KUKA KRL program: f1_Kuka_APT214T03S14.SRC

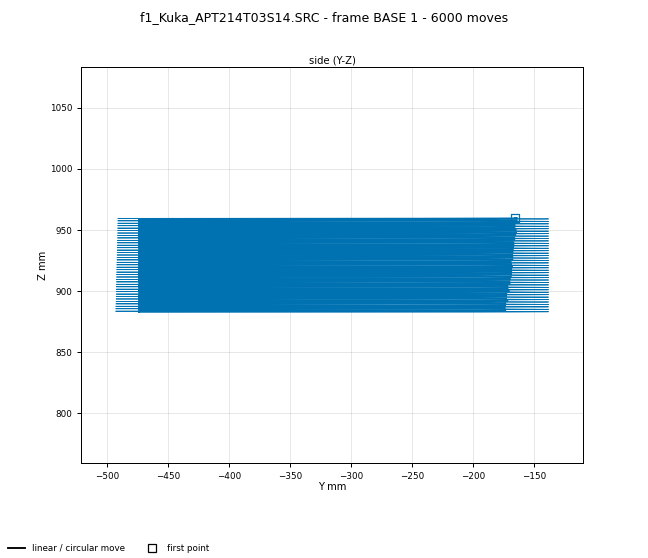
[picture p0: tool path of f1_Kuka_APT214T03S14.SRC in frame BASE 1, 6000 of 6001 moves have a stored position in this frame; points joined in program order, loops and branches not executed]
&ACCESS RVP
&REL 2
&PARAM TEMPLATE = C:\KRC\Roboter\Template\vorgabe
&PARAM EDITMASK = *
DEF f1_Kuka_APT214T03S14()


;FOLD INI;%{PE}%V3.2.0,%MKUKATPBASIS,%CINIT,%VCOMMON,%P
  ;FOLD BAS INI;%{E}%V3.2.0,%MKUKATPBASIS,%CINIT,%VINIT,%P
    GLOBAL INTERRUPT DECL 3 WHEN $STOPMESS==TRUE DO IR_STOPM ( )
    INTERRUPT ON 3
    BAS (#INITMOV,0 )
  ;ENDFOLD (BAS INI)
  ;FOLD USER INI;%{E}%V3.2.0,%MKUKATPUSER,%CINIT,%VINIT,%P
    ;Make your modifications here
  ;ENDFOLD (USER INI)
;ENDFOLD (INI)


;*** Make Null PTP Move
  PTP $pos_act

;*** Auto Load The Correct TOOL Data
  $tool=tool_data[3]

;*** Auto Load The Correct BASE Data
  $base=base_data[1]

  $ADVANCE = 5

;*** Restate Last Velocity
MMPM(30000.0)
SetRPM(6000)
LIN {X -0.031,Y -166.168,Z 960.065,A 0.000,B 0.000,C 90.000,E1 11.658} C_DIS
LIN {X 0.050,Y -163.859,Z 960.031,A 0.000,B 0.000,C 90.000,E1 5.511} C_DIS
LIN {X 0.017,Y -164.871,Z 959.968,A 0.000,B 0.000,C 90.000,E1 354.261} C_DIS
LIN {X -0.078,Y -167.650,Z 959.939,A 0.000,B 0.000,C 90.000,E1 349.050} C_DIS
LIN {X -0.007,Y -171.184,Z 959.915,A 0.000,B 0.000,C 90.000,E1 344.685} C_DIS
LIN {X 0.034,Y -175.840,Z 959.891,A 0.000,B 0.000,C 90.000,E1 340.369} C_DIS
LIN {X -0.004,Y -180.404,Z 959.872,A 0.000,B 0.000,C 90.000,E1 336.975} C_DIS
LIN {X 0.045,Y -185.731,Z 959.853,A 0.000,B 0.000,C 90.000,E1 333.589} C_DIS
LIN {X 0.060,Y -191.719,Z 959.835,A 0.000,B 0.000,C 90.000,E1 330.255} C_DIS
LIN {X -0.013,Y -198.321,Z 959.817,A 0.000,B 0.000,C 90.000,E1 326.993} C_DIS
LIN {X 0.015,Y -205.507,Z 959.799,A 0.000,B 0.000,C 90.000,E1 323.749} C_DIS
LIN {X -0.070,Y -214.244,Z 959.779,A 0.000,B 0.000,C 90.000,E1 320.194} C_DIS
LIN {X 0.036,Y -223.799,Z 959.759,A 0.000,B 0.000,C 90.000,E1 316.662} C_DIS
LIN {X -0.127,Y -232.037,Z 959.744,A 0.000,B 0.000,C 90.000,E1 314.028} C_DIS
LIN {X 0.056,Y -241.361,Z 959.730,A 0.000,B 0.000,C 90.000,E1 311.353} C_DIS
LIN {X 0.001,Y -250.281,Z 959.718,A 0.000,B 0.000,C 90.000,E1 309.152} C_DIS
LIN {X -0.109,Y -258.596,Z 959.707,A 0.000,B 0.000,C 90.000,E1 307.363} C_DIS
LIN {X 0.141,Y -271.571,Z 959.694,A 0.000,B 0.000,C 90.000,E1 304.818} C_DIS
LIN {X -0.058,Y -289.760,Z 959.676,A 0.000,B 0.000,C 90.000,E1 301.750} C_DIS
LIN {X -0.100,Y -304.933,Z 959.663,A 0.000,B 0.000,C 90.000,E1 299.411} C_DIS
LIN {X -0.098,Y -321.503,Z 959.651,A 0.000,B 0.000,C 90.000,E1 297.129} C_DIS
LIN {X -0.106,Y -334.635,Z 959.642,A 0.000,B 0.000,C 90.000,E1 295.540} C_DIS
LIN {X -0.116,Y -358.818,Z 959.627,A 0.000,B 0.000,C 90.000,E1 292.898} C_DIS
LIN {X -0.081,Y -377.767,Z 959.616,A 0.000,B 0.000,C 90.000,E1 290.972} C_DIS
LIN {X -0.056,Y -393.711,Z 959.608,A 0.000,B 0.000,C 90.000,E1 289.396} C_DIS
LIN {X -0.107,Y -404.139,Z 959.602,A 0.000,B 0.000,C 90.000,E1 288.362} C_DIS
LIN {X 0.117,Y -414.354,Z 959.596,A 0.000,B 0.000,C 90.000,E1 287.275} C_DIS
LIN {X 0.081,Y -424.254,Z 959.590,A 0.000,B 0.000,C 90.000,E1 286.205} C_DIS
LIN {X 0.005,Y -433.708,Z 959.584,A 0.000,B 0.000,C 90.000,E1 285.134} C_DIS
LIN {X 0.038,Y -442.447,Z 959.578,A 0.000,B 0.000,C 90.000,E1 284.064} C_DIS
LIN {X 0.069,Y -450.785,Z 959.572,A 0.000,B 0.000,C 90.000,E1 283.008} C_DIS
LIN {X 0.028,Y -460.710,Z 959.565,A 0.000,B 0.000,C 90.000,E1 281.715} C_DIS
LIN {X -0.184,Y -468.269,Z 959.559,A 0.000,B 0.000,C 90.000,E1 280.715} C_DIS
LIN {X 0.202,Y -473.450,Z 959.555,A 0.000,B 0.000,C 90.000,E1 279.905} C_DIS
LIN {X 0.180,Y -478.073,Z 959.551,A 0.000,B 0.000,C 90.000,E1 279.151} C_DIS
LIN {X 0.195,Y -481.999,Z 959.547,A 0.000,B 0.000,C 90.000,E1 278.398} C_DIS
LIN {X -0.115,Y -484.263,Z 959.544,A 0.000,B 0.000,C 90.000,E1 277.936} C_DIS
LIN {X 0.131,Y -486.237,Z 959.541,A 0.000,B 0.000,C 90.000,E1 277.409} C_DIS
LIN {X -0.165,Y -487.852,Z 959.539,A 0.000,B 0.000,C 90.000,E1 276.947} C_DIS
LIN {X 0.034,Y -489.159,Z 959.536,A 0.000,B 0.000,C 90.000,E1 276.429} C_DIS
LIN {X 0.244,Y -490.135,Z 959.533,A 0.000,B 0.000,C 90.000,E1 275.910} C_DIS
LIN {X -0.074,Y -490.762,Z 959.530,A 0.000,B 0.000,C 90.000,E1 275.454} C_DIS
LIN {X 0.152,Y -491.016,Z 959.528,A 0.000,B 0.000,C 90.000,E1 274.935} C_DIS
LIN {X -0.111,Y -490.869,Z 959.525,A 0.000,B 0.000,C 90.000,E1 274.473} C_DIS
LIN {X 0.114,Y -490.251,Z 959.522,A 0.000,B 0.000,C 90.000,E1 273.955} C_DIS
LIN {X -0.183,Y -489.140,Z 959.519,A 0.000,B 0.000,C 90.000,E1 273.498} C_DIS
LIN {X 0.034,Y -487.440,Z 959.517,A 0.000,B 0.000,C 90.000,E1 272.980} C_DIS
LIN {X 0.217,Y -485.143,Z 959.514,A 0.000,B 0.000,C 90.000,E1 272.465} C_DIS
LIN {X -0.095,Y -482.097,Z 959.511,A 0.000,B 0.000,C 90.000,E1 272.007} C_DIS
LIN {X 0.074,Y -478.192,Z 959.508,A 0.000,B 0.000,C 90.000,E1 271.489} C_DIS
LIN {X 0.207,Y -473.231,Z 959.506,A 0.000,B 0.000,C 90.000,E1 270.974} C_DIS
LIN {X 0.022,Y -467.466,Z 959.503,A 0.000,B 0.000,C 90.000,E1 270.516} C_DIS
LIN {X -0.191,Y -461.347,Z 959.500,A 0.000,B 0.000,C 90.000,E1 270.115} C_DIS
LIN {X -0.006,Y -454.864,Z 959.498,A 0.000,B 0.000,C 90.000,E1 269.714} C_DIS
LIN {X 0.154,Y -448.019,Z 959.497,A 0.000,B 0.000,C 90.000,E1 269.370} C_DIS
LIN {X -0.150,Y -441.116,Z 959.495,A 0.000,B 0.000,C 90.000,E1 269.141} C_DIS
LIN {X -0.111,Y -433.920,Z 959.494,A 0.000,B 0.000,C 90.000,E1 268.912} C_DIS
LIN {X -0.201,Y -426.014,Z 959.493,A 0.000,B 0.000,C 90.000,E1 268.740} C_DIS
LIN {X 0.015,Y -417.851,Z 959.492,A 0.000,B 0.000,C 90.000,E1 268.568} C_DIS
LIN {X -0.140,Y -410.678,Z 959.492,A 0.000,B 0.000,C 90.000,E1 268.511} C_DIS
LIN {X -0.033,Y -402.201,Z 959.491,A 0.000,B 0.000,C 90.000,E1 268.453} C_DIS
LIN {X -0.040,Y -181.202,Z 959.491,A 0.000,B 0.000,C 90.000,E1 268.453} C_DIS
LIN {X 0.070,Y -180.868,Z 959.472,A 0.000,B 0.000,C 90.000,E1 265.008} C_DIS
LIN {X -0.054,Y -178.983,Z 959.444,A 0.000,B 0.000,C 90.000,E1 259.982} C_DIS
LIN {X -0.042,Y -177.958,Z 959.435,A 0.000,B 0.000,C 90.000,E1 258.285} C_DIS
LIN {X -0.022,Y -175.600,Z 959.411,A 0.000,B 0.000,C 90.000,E1 254.031} C_DIS
LIN {X -0.009,Y -172.324,Z 959.388,A 0.000,B 0.000,C 90.000,E1 249.752} C_DIS
LIN {X -0.031,Y -171.801,Z 959.383,A 0.000,B 0.000,C 90.000,E1 248.901} C_DIS
LIN {X 0.006,Y -169.476,Z 959.368,A 0.000,B 0.000,C 90.000,E1 246.305} C_DIS
LIN {X -0.087,Y -166.803,Z 959.349,A 0.000,B 0.000,C 90.000,E1 242.871} C_DIS
LIN {X 0.056,Y -162.783,Z 959.325,A 0.000,B 0.000,C 90.000,E1 238.456} C_DIS
LIN {X 0.032,Y -161.472,Z 959.315,A 0.000,B 0.000,C 90.000,E1 236.707} C_DIS
LIN {X 0.073,Y -157.467,Z 959.291,A 0.000,B 0.000,C 90.000,E1 232.271} C_DIS
LIN {X 0.005,Y -155.481,Z 959.276,A 0.000,B 0.000,C 90.000,E1 229.622} C_DIS
LIN {X -0.062,Y -151.789,Z 959.251,A 0.000,B 0.000,C 90.000,E1 225.162} C_DIS
LIN {X -0.048,Y -149.998,Z 959.236,A 0.000,B 0.000,C 90.000,E1 222.447} C_DIS
LIN {X -0.017,Y -146.827,Z 959.210,A 0.000,B 0.000,C 90.000,E1 217.890} C_DIS
LIN {X -0.030,Y -145.407,Z 959.195,A 0.000,B 0.000,C 90.000,E1 215.152} C_DIS
LIN {X 0.005,Y -142.839,Z 959.170,A 0.000,B 0.000,C 90.000,E1 210.541} C_DIS
LIN {X -0.064,Y -141.452,Z 959.149,A 0.000,B 0.000,C 90.000,E1 206.873} C_DIS
LIN {X -0.025,Y -139.372,Z 959.113,A 0.000,B 0.000,C 90.000,E1 200.355} C_DIS
LIN {X -0.082,Y -138.821,Z 959.097,A 0.000,B 0.000,C 90.000,E1 197.583} C_DIS
LIN {X 0.007,Y -138.352,Z 959.056,A 0.000,B 0.000,C 90.000,E1 190.074} C_DIS
LIN {X -0.021,Y -139.534,Z 959.004,A 0.000,B 0.000,C 90.000,E1 180.745} C_DIS
LIN {X 0.072,Y -141.217,Z 958.973,A 0.000,B 0.000,C 90.000,E1 175.122} C_DIS
LIN {X 0.032,Y -142.591,Z 958.958,A 0.000,B 0.000,C 90.000,E1 172.356} C_DIS
LIN {X -0.014,Y -144.891,Z 958.932,A 0.000,B 0.000,C 90.000,E1 167.757} C_DIS
LIN {X -0.062,Y -147.519,Z 958.912,A 0.000,B 0.000,C 90.000,E1 164.102} C_DIS
LIN {X 0.013,Y -150.113,Z 958.891,A 0.000,B 0.000,C 90.000,E1 160.423} C_DIS
LIN {X 0.025,Y -153.473,Z 958.871,A 0.000,B 0.000,C 90.000,E1 156.794} C_DIS
LIN {X 0.015,Y -157.838,Z 958.846,A 0.000,B 0.000,C 90.000,E1 152.308} C_DIS
LIN {X 0.046,Y -162.122,Z 958.826,A 0.000,B 0.000,C 90.000,E1 148.742} C_DIS
LIN {X -0.069,Y -166.324,Z 958.807,A 0.000,B 0.000,C 90.000,E1 145.261} C_DIS
LIN {X 0.032,Y -171.341,Z 958.788,A 0.000,B 0.000,C 90.000,E1 141.743} C_DIS
LIN {X -0.041,Y -176.244,Z 958.768,A 0.000,B 0.000,C 90.000,E1 138.324} C_DIS
LIN {X 0.079,Y -180.525,Z 958.754,A 0.000,B 0.000,C 90.000,E1 135.729} C_DIS
LIN {X 0.059,Y -185.928,Z 958.735,A 0.000,B 0.000,C 90.000,E1 132.366} C_DIS
LIN {X -0.007,Y -190.558,Z 958.722,A 0.000,B 0.000,C 90.000,E1 129.886} C_DIS
LIN {X 0.020,Y -194.806,Z 958.708,A 0.000,B 0.000,C 90.000,E1 127.397} C_DIS
LIN {X -0.006,Y -297.968,Z 958.708,A 0.000,B 0.000,C 90.000,E1 127.397} C_DIS
LIN {X -0.109,Y -300.519,Z 958.707,A 0.000,B 0.000,C 90.000,E1 127.363} C_DIS
LIN {X -0.014,Y -304.144,Z 958.706,A 0.000,B 0.000,C 90.000,E1 127.156} C_DIS
LIN {X 0.086,Y -306.383,Z 958.705,A 0.000,B 0.000,C 90.000,E1 126.950} C_DIS
LIN {X 0.037,Y -309.504,Z 958.703,A 0.000,B 0.000,C 90.000,E1 126.583} C_DIS
LIN {X -0.163,Y -311.442,Z 958.701,A 0.000,B 0.000,C 90.000,E1 126.297} C_DIS
LIN {X 0.072,Y -312.952,Z 958.700,A 0.000,B 0.000,C 90.000,E1 125.931} C_DIS
LIN {X -0.087,Y -315.137,Z 958.696,A 0.000,B 0.000,C 90.000,E1 125.311} C_DIS
LIN {X 0.037,Y -325.779,Z 958.678,A 0.000,B 0.000,C 90.000,E1 122.084} C_DIS
LIN {X -0.132,Y -336.713,Z 958.663,A 0.000,B 0.000,C 90.000,E1 119.283} C_DIS
LIN {X -0.033,Y -349.037,Z 958.647,A 0.000,B 0.000,C 90.000,E1 116.488} C_DIS
LIN {X -0.038,Y -362.857,Z 958.632,A 0.000,B 0.000,C 90.000,E1 113.770} C_DIS
LIN {X -0.051,Y -376.497,Z 958.619,A 0.000,B 0.000,C 90.000,E1 111.408} C_DIS
LIN {X 0.003,Y -391.515,Z 958.606,A 0.000,B 0.000,C 90.000,E1 109.087} C_DIS
LIN {X -0.201,Y -408.016,Z 958.594,A 0.000,B 0.000,C 90.000,E1 106.858} C_DIS
LIN {X -0.131,Y -426.122,Z 958.581,A 0.000,B 0.000,C 90.000,E1 104.647} C_DIS
LIN {X -0.199,Y -445.757,Z 958.570,A 0.000,B 0.000,C 90.000,E1 102.535} C_DIS
LIN {X 0.059,Y -466.092,Z 958.559,A 0.000,B 0.000,C 90.000,E1 100.546} C_DIS
LIN {X 0.072,Y -468.438,Z 958.557,A 0.000,B 0.000,C 90.000,E1 100.310} C_DIS
LIN {X -0.026,Y -470.296,Z 958.556,A 0.000,B 0.000,C 90.000,E1 100.074} C_DIS
LIN {X -0.207,Y -471.699,Z 958.555,A 0.000,B 0.000,C 90.000,E1 99.849} C_DIS
LIN {X -0.031,Y -473.539,Z 958.552,A 0.000,B 0.000,C 90.000,E1 99.321} C_DIS
LIN {X 0.077,Y -474.283,Z 958.549,A 0.000,B 0.000,C 90.000,E1 98.803} C_DIS
LIN {X 0.268,Y -474.059,Z 958.546,A 0.000,B 0.000,C 90.000,E1 98.276} C_DIS
LIN {X -0.077,Y -472.835,Z 958.543,A 0.000,B 0.000,C 90.000,E1 97.814} C_DIS
LIN {X 0.188,Y -471.792,Z 958.542,A 0.000,B 0.000,C 90.000,E1 97.530} C_DIS
LIN {X 0.047,Y -470.392,Z 958.541,A 0.000,B 0.000,C 90.000,E1 97.296} C_DIS
LIN {X 0.100,Y -458.658,Z 958.531,A 0.000,B 0.000,C 90.000,E1 95.511} C_DIS
LIN {X 0.121,Y -445.384,Z 958.519,A 0.000,B 0.000,C 90.000,E1 93.440} C_DIS
LIN {X 0.105,Y -428.779,Z 958.505,A 0.000,B 0.000,C 90.000,E1 90.802} C_DIS
LIN {X 0.128,Y -411.902,Z 958.488,A 0.000,B 0.000,C 90.000,E1 87.822} C_DIS
LIN {X 0.175,Y -402.774,Z 958.479,A 0.000,B 0.000,C 90.000,E1 86.159} C_DIS
LIN {X 0.131,Y -392.001,Z 958.468,A 0.000,B 0.000,C 90.000,E1 84.204} C_DIS
LIN {X -0.067,Y -382.677,Z 958.458,A 0.000,B 0.000,C 90.000,E1 82.527} C_DIS
LIN {X -0.047,Y -373.069,Z 958.449,A 0.000,B 0.000,C 90.000,E1 80.792} C_DIS
LIN {X -0.148,Y -363.193,Z 958.439,A 0.000,B 0.000,C 90.000,E1 79.050} C_DIS
LIN {X 0.066,Y -353.138,Z 958.429,A 0.000,B 0.000,C 90.000,E1 77.229} C_DIS
LIN {X -0.090,Y -338.180,Z 958.414,A 0.000,B 0.000,C 90.000,E1 74.519} C_DIS
LIN {X 0.039,Y -324.200,Z 958.398,A 0.000,B 0.000,C 90.000,E1 71.692} C_DIS
LIN {X -0.036,Y -312.152,Z 958.384,A 0.000,B 0.000,C 90.000,E1 69.156} C_DIS
LIN {X 0.027,Y -301.623,Z 958.372,A 0.000,B 0.000,C 90.000,E1 66.869} C_DIS
LIN {X 0.094,Y -291.227,Z 958.359,A 0.000,B 0.000,C 90.000,E1 64.537} C_DIS
LIN {X 0.061,Y -280.913,Z 958.346,A 0.000,B 0.000,C 90.000,E1 62.180} C_DIS
LIN {X -0.046,Y -270.635,Z 958.332,A 0.000,B 0.000,C 90.000,E1 59.793} C_DIS
LIN {X 0.050,Y -259.319,Z 958.317,A 0.000,B 0.000,C 90.000,E1 56.962} C_DIS
LIN {X -0.049,Y -247.134,Z 958.299,A 0.000,B 0.000,C 90.000,E1 53.749} C_DIS
LIN {X -0.049,Y -235.992,Z 958.280,A 0.000,B 0.000,C 90.000,E1 50.436} C_DIS
LIN {X 0.050,Y -225.633,Z 958.261,A 0.000,B 0.000,C 90.000,E1 47.025} C_DIS
LIN {X 0.088,Y -217.040,Z 958.244,A 0.000,B 0.000,C 90.000,E1 43.947} C_DIS
LIN {X -0.045,Y -208.949,Z 958.227,A 0.000,B 0.000,C 90.000,E1 40.862} C_DIS
LIN {X -0.029,Y -201.480,Z 958.209,A 0.000,B 0.000,C 90.000,E1 37.684} C_DIS
LIN {X -0.008,Y -194.630,Z 958.191,A 0.000,B 0.000,C 90.000,E1 34.452} C_DIS
LIN {X -0.013,Y -188.415,Z 958.173,A 0.000,B 0.000,C 90.000,E1 31.180} C_DIS
LIN {X 0.030,Y -182.953,Z 958.155,A 0.000,B 0.000,C 90.000,E1 27.847} C_DIS
LIN {X -0.062,Y -178.106,Z 958.136,A 0.000,B 0.000,C 90.000,E1 24.515} C_DIS
LIN {X -0.015,Y -173.074,Z 958.112,A 0.000,B 0.000,C 90.000,E1 20.248} C_DIS
LIN {X -0.032,Y -169.140,Z 958.089,A 0.000,B 0.000,C 90.000,E1 15.953} C_DIS
LIN {X 0.039,Y -166.285,Z 958.064,A 0.000,B 0.000,C 90.000,E1 11.591} C_DIS
LIN {X -0.070,Y -163.987,Z 958.030,A 0.000,B 0.000,C 90.000,E1 5.511} C_DIS
LIN {X 0.023,Y -165.053,Z 957.968,A 0.000,B 0.000,C 90.000,E1 354.261} C_DIS
LIN {X -0.065,Y -167.841,Z 957.939,A 0.000,B 0.000,C 90.000,E1 349.050} C_DIS
LIN {X -0.032,Y -171.390,Z 957.915,A 0.000,B 0.000,C 90.000,E1 344.700} C_DIS
LIN {X 0.061,Y -176.062,Z 957.891,A 0.000,B 0.000,C 90.000,E1 340.369} C_DIS
LIN {X 0.028,Y -180.646,Z 957.872,A 0.000,B 0.000,C 90.000,E1 336.975} C_DIS
LIN {X -0.082,Y -185.957,Z 957.853,A 0.000,B 0.000,C 90.000,E1 333.640} C_DIS
LIN {X 0.012,Y -191.932,Z 957.835,A 0.000,B 0.000,C 90.000,E1 330.284} C_DIS
LIN {X 0.040,Y -198.523,Z 957.817,A 0.000,B 0.000,C 90.000,E1 326.993} C_DIS
LIN {X -0.045,Y -205.728,Z 957.799,A 0.000,B 0.000,C 90.000,E1 323.783} C_DIS
LIN {X -0.039,Y -213.425,Z 957.781,A 0.000,B 0.000,C 90.000,E1 320.598} C_DIS
LIN {X 0.041,Y -222.894,Z 957.762,A 0.000,B 0.000,C 90.000,E1 317.067} C_DIS
LIN {X -0.042,Y -232.250,Z 957.745,A 0.000,B 0.000,C 90.000,E1 314.028} C_DIS
LIN {X 0.133,Y -242.974,Z 957.728,A 0.000,B 0.000,C 90.000,E1 310.987} C_DIS
LIN {X -0.081,Y -252.062,Z 957.716,A 0.000,B 0.000,C 90.000,E1 308.830} C_DIS
LIN {X 0.001,Y -258.762,Z 957.708,A 0.000,B 0.000,C 90.000,E1 307.363} C_DIS
LIN {X -0.120,Y -271.661,Z 957.694,A 0.000,B 0.000,C 90.000,E1 304.898} C_DIS
LIN {X 0.070,Y -289.797,Z 957.676,A 0.000,B 0.000,C 90.000,E1 301.750} C_DIS
LIN {X 0.035,Y -304.932,Z 957.663,A 0.000,B 0.000,C 90.000,E1 299.411} C_DIS
LIN {X 0.044,Y -321.401,Z 957.651,A 0.000,B 0.000,C 90.000,E1 297.129} C_DIS
LIN {X 0.062,Y -333.998,Z 957.642,A 0.000,B 0.000,C 90.000,E1 295.591} C_DIS
LIN {X 0.025,Y -358.052,Z 957.628,A 0.000,B 0.000,C 90.000,E1 292.950} C_DIS
LIN {X -0.067,Y -379.492,Z 957.615,A 0.000,B 0.000,C 90.000,E1 290.791} C_DIS
LIN {X 0.028,Y -392.885,Z 957.608,A 0.000,B 0.000,C 90.000,E1 289.450} C_DIS
LIN {X -0.063,Y -403.354,Z 957.602,A 0.000,B 0.000,C 90.000,E1 288.417} C_DIS
LIN {X 0.130,Y -413.596,Z 957.596,A 0.000,B 0.000,C 90.000,E1 287.330} C_DIS
LIN {X 0.100,Y -423.566,Z 957.590,A 0.000,B 0.000,C 90.000,E1 286.260} C_DIS
LIN {X 0.017,Y -433.028,Z 957.584,A 0.000,B 0.000,C 90.000,E1 285.190} C_DIS
LIN {X 0.040,Y -441.816,Z 957.578,A 0.000,B 0.000,C 90.000,E1 284.120} C_DIS
LIN {X -0.135,Y -452.195,Z 957.571,A 0.000,B 0.000,C 90.000,E1 282.827} C_DIS
LIN {X -0.169,Y -462.102,Z 957.564,A 0.000,B 0.000,C 90.000,E1 281.535} C_DIS
LIN {X 0.003,Y -469.556,Z 957.558,A 0.000,B 0.000,C 90.000,E1 280.489} C_DIS
LIN {X 0.026,Y -474.604,Z 957.554,A 0.000,B 0.000,C 90.000,E1 279.726} C_DIS
LIN {X 0.005,Y -479.128,Z 957.550,A 0.000,B 0.000,C 90.000,E1 278.973} C_DIS
LIN {X 0.029,Y -482.897,Z 957.546,A 0.000,B 0.000,C 90.000,E1 278.219} C_DIS
LIN {X 0.082,Y -486.004,Z 957.542,A 0.000,B 0.000,C 90.000,E1 277.466} C_DIS
LIN {X -0.217,Y -487.679,Z 957.539,A 0.000,B 0.000,C 90.000,E1 277.004} C_DIS
LIN {X -0.019,Y -489.027,Z 957.536,A 0.000,B 0.000,C 90.000,E1 276.486} C_DIS
LIN {X 0.189,Y -490.059,Z 957.533,A 0.000,B 0.000,C 90.000,E1 275.967} C_DIS
LIN {X -0.130,Y -490.734,Z 957.531,A 0.000,B 0.000,C 90.000,E1 275.511} C_DIS
LIN {X 0.094,Y -491.036,Z 957.528,A 0.000,B 0.000,C 90.000,E1 274.992} C_DIS
LIN {X -0.168,Y -490.957,Z 957.525,A 0.000,B 0.000,C 90.000,E1 274.531} C_DIS
LIN {X 0.056,Y -490.405,Z 957.522,A 0.000,B 0.000,C 90.000,E1 274.012} C_DIS
LIN {X -0.241,Y -489.317,Z 957.520,A 0.000,B 0.000,C 90.000,E1 273.555} C_DIS
LIN {X -0.022,Y -487.729,Z 957.517,A 0.000,B 0.000,C 90.000,E1 273.037} C_DIS
LIN {X -0.174,Y -486.739,Z 957.516,A 0.000,B 0.000,C 90.000,E1 272.808} C_DIS
LIN {X 0.006,Y -484.152,Z 957.513,A 0.000,B 0.000,C 90.000,E1 272.293} C_DIS
LIN {X 0.187,Y -480.765,Z 957.510,A 0.000,B 0.000,C 90.000,E1 271.776} C_DIS
LIN {X -0.146,Y -476.527,Z 957.507,A 0.000,B 0.000,C 90.000,E1 271.318} C_DIS
LIN {X 0.044,Y -471.215,Z 957.504,A 0.000,B 0.000,C 90.000,E1 270.802} C_DIS
LIN {X 0.021,Y -465.321,Z 957.502,A 0.000,B 0.000,C 90.000,E1 270.344} C_DIS
LIN {X -0.054,Y -459.128,Z 957.500,A 0.000,B 0.000,C 90.000,E1 269.943} C_DIS
LIN {X -0.164,Y -452.517,Z 957.498,A 0.000,B 0.000,C 90.000,E1 269.599} C_DIS
LIN {X 0.141,Y -445.677,Z 957.496,A 0.000,B 0.000,C 90.000,E1 269.255} C_DIS
LIN {X -0.057,Y -438.526,Z 957.495,A 0.000,B 0.000,C 90.000,E1 269.026} C_DIS
LIN {X 0.078,Y -431.034,Z 957.493,A 0.000,B 0.000,C 90.000,E1 268.797} C_DIS
LIN {X 0.090,Y -423.172,Z 957.492,A 0.000,B 0.000,C 90.000,E1 268.625} C_DIS
LIN {X -0.031,Y -414.503,Z 957.492,A 0.000,B 0.000,C 90.000,E1 268.511} C_DIS
LIN {X -0.027,Y -407.110,Z 957.491,A 0.000,B 0.000,C 90.000,E1 268.453} C_DIS
LIN {X -0.140,Y -402.934,Z 957.491,A 0.000,B 0.000,C 90.000,E1 268.453} C_DIS
LIN {X -0.088,Y -181.199,Z 957.491,A 0.000,B 0.000,C 90.000,E1 268.453} C_DIS
LIN {X 0.022,Y -180.865,Z 957.472,A 0.000,B 0.000,C 90.000,E1 265.008} C_DIS
LIN {X 0.075,Y -178.979,Z 957.444,A 0.000,B 0.000,C 90.000,E1 259.926} C_DIS
LIN {X 0.085,Y -177.948,Z 957.435,A 0.000,B 0.000,C 90.000,E1 258.229} C_DIS
LIN {X -0.069,Y -175.589,Z 957.411,A 0.000,B 0.000,C 90.000,E1 254.031} C_DIS
LIN {X -0.057,Y -172.315,Z 957.387,A 0.000,B 0.000,C 90.000,E1 249.752} C_DIS
LIN {X -0.078,Y -171.792,Z 957.383,A 0.000,B 0.000,C 90.000,E1 248.901} C_DIS
LIN {X -0.040,Y -169.462,Z 957.368,A 0.000,B 0.000,C 90.000,E1 246.305} C_DIS
LIN {X 0.016,Y -166.791,Z 957.349,A 0.000,B 0.000,C 90.000,E1 242.820} C_DIS
LIN {X 0.011,Y -162.771,Z 957.325,A 0.000,B 0.000,C 90.000,E1 238.456} C_DIS
LIN {X -0.012,Y -161.460,Z 957.315,A 0.000,B 0.000,C 90.000,E1 236.707} C_DIS
LIN {X 0.029,Y -157.454,Z 957.290,A 0.000,B 0.000,C 90.000,E1 232.271} C_DIS
LIN {X -0.038,Y -155.465,Z 957.276,A 0.000,B 0.000,C 90.000,E1 229.622} C_DIS
LIN {X 0.003,Y -151.779,Z 957.251,A 0.000,B 0.000,C 90.000,E1 225.121} C_DIS
LIN {X 0.019,Y -149.984,Z 957.236,A 0.000,B 0.000,C 90.000,E1 222.405} C_DIS
LIN {X -0.059,Y -146.817,Z 957.210,A 0.000,B 0.000,C 90.000,E1 217.890} C_DIS
LIN {X 0.046,Y -145.396,Z 957.195,A 0.000,B 0.000,C 90.000,E1 215.105} C_DIS
LIN {X -0.036,Y -142.832,Z 957.170,A 0.000,B 0.000,C 90.000,E1 210.541} C_DIS
LIN {X 0.021,Y -141.443,Z 957.149,A 0.000,B 0.000,C 90.000,E1 206.821} C_DIS
LIN {X 0.065,Y -139.369,Z 957.113,A 0.000,B 0.000,C 90.000,E1 200.301} C_DIS
LIN {X 0.051,Y -138.817,Z 957.097,A 0.000,B 0.000,C 90.000,E1 197.511} C_DIS
LIN {X -0.035,Y -138.352,Z 957.056,A 0.000,B 0.000,C 90.000,E1 190.074} C_DIS
LIN {X -0.062,Y -139.536,Z 957.004,A 0.000,B 0.000,C 90.000,E1 180.745} C_DIS
LIN {X 0.032,Y -141.225,Z 956.973,A 0.000,B 0.000,C 90.000,E1 175.122} C_DIS
LIN {X -0.010,Y -142.596,Z 956.958,A 0.000,B 0.000,C 90.000,E1 172.356} C_DIS
LIN {X -0.056,Y -144.901,Z 956.932,A 0.000,B 0.000,C 90.000,E1 167.757} C_DIS
LIN {X 0.038,Y -147.529,Z 956.911,A 0.000,B 0.000,C 90.000,E1 164.047} C_DIS
LIN {X -0.030,Y -150.127,Z 956.891,A 0.000,B 0.000,C 90.000,E1 160.423} C_DIS
LIN {X -0.019,Y -153.491,Z 956.871,A 0.000,B 0.000,C 90.000,E1 156.794} C_DIS
LIN {X 0.045,Y -157.855,Z 956.846,A 0.000,B 0.000,C 90.000,E1 152.281} C_DIS
LIN {X 0.001,Y -162.141,Z 956.826,A 0.000,B 0.000,C 90.000,E1 148.742} C_DIS
LIN {X -0.021,Y -166.345,Z 956.807,A 0.000,B 0.000,C 90.000,E1 145.229} C_DIS
LIN {X -0.015,Y -171.362,Z 956.787,A 0.000,B 0.000,C 90.000,E1 141.743} C_DIS
LIN {X -0.088,Y -176.268,Z 956.768,A 0.000,B 0.000,C 90.000,E1 138.324} C_DIS
LIN {X 0.031,Y -180.552,Z 956.754,A 0.000,B 0.000,C 90.000,E1 135.729} C_DIS
LIN {X 0.010,Y -185.954,Z 956.735,A 0.000,B 0.000,C 90.000,E1 132.366} C_DIS
LIN {X 0.066,Y -190.586,Z 956.721,A 0.000,B 0.000,C 90.000,E1 129.850} C_DIS
LIN {X -0.022,Y -194.746,Z 956.708,A 0.000,B 0.000,C 90.000,E1 127.443} C_DIS
LIN {X -0.088,Y -297.857,Z 956.708,A 0.000,B 0.000,C 90.000,E1 127.443} C_DIS
LIN {X -0.011,Y -299.609,Z 956.708,A 0.000,B 0.000,C 90.000,E1 127.397} C_DIS
LIN {X 0.080,Y -302.988,Z 956.707,A 0.000,B 0.000,C 90.000,E1 127.237} C_DIS
LIN {X -0.049,Y -306.366,Z 956.706,A 0.000,B 0.000,C 90.000,E1 126.996} C_DIS
LIN {X 0.110,Y -310.028,Z 956.703,A 0.000,B 0.000,C 90.000,E1 126.503} C_DIS
LIN {X -0.111,Y -311.840,Z 956.701,A 0.000,B 0.000,C 90.000,E1 126.217} C_DIS
LIN {X -0.081,Y -313.256,Z 956.699,A 0.000,B 0.000,C 90.000,E1 125.884} C_DIS
LIN {X -0.018,Y -324.881,Z 956.680,A 0.000,B 0.000,C 90.000,E1 122.339} C_DIS
LIN {X 0.067,Y -335.703,Z 956.664,A 0.000,B 0.000,C 90.000,E1 119.489} C_DIS
LIN {X -0.156,Y -347.901,Z 956.648,A 0.000,B 0.000,C 90.000,E1 116.744} C_DIS
LIN {X -0.056,Y -361.590,Z 956.633,A 0.000,B 0.000,C 90.000,E1 114.003} C_DIS
LIN {X -0.111,Y -375.105,Z 956.620,A 0.000,B 0.000,C 90.000,E1 111.642} C_DIS
LIN {X -0.103,Y -389.985,Z 956.607,A 0.000,B 0.000,C 90.000,E1 109.322} C_DIS
LIN {X 0.033,Y -406.340,Z 956.595,A 0.000,B 0.000,C 90.000,E1 107.040} C_DIS
LIN {X 0.074,Y -424.286,Z 956.582,A 0.000,B 0.000,C 90.000,E1 104.828} C_DIS
LIN {X 0.018,Y -443.817,Z 956.571,A 0.000,B 0.000,C 90.000,E1 102.703} C_DIS
LIN {X 0.144,Y -464.099,Z 956.560,A 0.000,B 0.000,C 90.000,E1 100.715} C_DIS
LIN {X 0.077,Y -466.659,Z 956.558,A 0.000,B 0.000,C 90.000,E1 100.489} C_DIS
LIN {X 0.095,Y -468.866,Z 956.557,A 0.000,B 0.000,C 90.000,E1 100.254} C_DIS
LIN {X -0.058,Y -470.658,Z 956.556,A 0.000,B 0.000,C 90.000,E1 100.018} C_DIS
LIN {X 0.251,Y -472.005,Z 956.554,A 0.000,B 0.000,C 90.000,E1 99.726} C_DIS
LIN {X -0.115,Y -473.691,Z 956.551,A 0.000,B 0.000,C 90.000,E1 99.265} C_DIS
LIN {X -0.004,Y -474.311,Z 956.549,A 0.000,B 0.000,C 90.000,E1 98.746} C_DIS
LIN {X 0.188,Y -473.964,Z 956.546,A 0.000,B 0.000,C 90.000,E1 98.219} C_DIS
LIN {X -0.156,Y -472.605,Z 956.543,A 0.000,B 0.000,C 90.000,E1 97.757} C_DIS
LIN {X 0.109,Y -471.478,Z 956.542,A 0.000,B 0.000,C 90.000,E1 97.473} C_DIS
LIN {X 0.079,Y -466.628,Z 956.537,A 0.000,B 0.000,C 90.000,E1 96.720} C_DIS
LIN {X -0.131,Y -453.282,Z 956.526,A 0.000,B 0.000,C 90.000,E1 94.702} C_DIS
LIN {X -0.191,Y -443.341,Z 956.517,A 0.000,B 0.000,C 90.000,E1 93.151} C_DIS
LIN {X 0.116,Y -422.154,Z 956.498,A 0.000,B 0.000,C 90.000,E1 89.656} C_DIS
LIN {X 0.109,Y -410.054,Z 956.486,A 0.000,B 0.000,C 90.000,E1 87.478} C_DIS
LIN {X 0.147,Y -400.864,Z 956.477,A 0.000,B 0.000,C 90.000,E1 85.812} C_DIS
LIN {X 0.078,Y -390.096,Z 956.466,A 0.000,B 0.000,C 90.000,E1 83.856} C_DIS
LIN {X -0.200,Y -380.695,Z 956.456,A 0.000,B 0.000,C 90.000,E1 82.186} C_DIS
LIN {X -0.161,Y -371.062,Z 956.447,A 0.000,B 0.000,C 90.000,E1 80.443} C_DIS
LIN {X 0.099,Y -359.466,Z 956.435,A 0.000,B 0.000,C 90.000,E1 78.342} C_DIS
LIN {X -0.180,Y -349.322,Z 956.425,A 0.000,B 0.000,C 90.000,E1 76.589} C_DIS
LIN {X -0.064,Y -331.473,Z 956.407,A 0.000,B 0.000,C 90.000,E1 73.196} C_DIS
LIN {X -0.056,Y -319.288,Z 956.393,A 0.000,B 0.000,C 90.000,E1 70.678} C_DIS
LIN {X 0.046,Y -308.795,Z 956.380,A 0.000,B 0.000,C 90.000,E1 68.411} C_DIS
LIN {X 0.037,Y -296.794,Z 956.366,A 0.000,B 0.000,C 90.000,E1 65.793} C_DIS
LIN {X 0.006,Y -286.426,Z 956.353,A 0.000,B 0.000,C 90.000,E1 63.461} C_DIS
LIN {X 0.126,Y -276.118,Z 956.339,A 0.000,B 0.000,C 90.000,E1 61.051} C_DIS
LIN {X -0.009,Y -263.146,Z 956.322,A 0.000,B 0.000,C 90.000,E1 57.946} C_DIS
LIN {X -0.017,Y -250.718,Z 956.304,A 0.000,B 0.000,C 90.000,E1 54.736} C_DIS
LIN {X -0.059,Y -239.288,Z 956.286,A 0.000,B 0.000,C 90.000,E1 51.457} C_DIS
LIN {X -0.014,Y -228.743,Z 956.267,A 0.000,B 0.000,C 90.000,E1 48.081} C_DIS
LIN {X 0.026,Y -218.872,Z 956.248,A 0.000,B 0.000,C 90.000,E1 44.636} C_DIS
LIN {X 0.073,Y -210.709,Z 956.231,A 0.000,B 0.000,C 90.000,E1 41.515} C_DIS
LIN {X -0.036,Y -203.115,Z 956.213,A 0.000,B 0.000,C 90.000,E1 38.382} C_DIS
LIN {X 0.023,Y -196.174,Z 956.195,A 0.000,B 0.000,C 90.000,E1 35.152} C_DIS
LIN {X 0.057,Y -189.839,Z 956.177,A 0.000,B 0.000,C 90.000,E1 31.878} C_DIS
LIN {X 0.068,Y -184.229,Z 956.159,A 0.000,B 0.000,C 90.000,E1 28.565} C_DIS
LIN {X 0.086,Y -179.250,Z 956.140,A 0.000,B 0.000,C 90.000,E1 25.207} C_DIS
LIN {X 0.005,Y -175.027,Z 956.121,A 0.000,B 0.000,C 90.000,E1 21.844} C_DIS
LIN {X 0.021,Y -171.414,Z 956.102,A 0.000,B 0.000,C 90.000,E1 18.417} C_DIS
LIN {X -0.035,Y -167.950,Z 956.078,A 0.000,B 0.000,C 90.000,E1 14.120} C_DIS
LIN {X 0.073,Y -165.149,Z 956.049,A 0.000,B 0.000,C 90.000,E1 8.859} C_DIS
LIN {X -0.015,Y -166.012,Z 955.958,A 0.000,B 0.000,C 90.000,E1 352.527} C_DIS
LIN {X -0.032,Y -168.673,Z 955.934,A 0.000,B 0.000,C 90.000,E1 348.173} C_DIS
LIN {X -0.051,Y -172.468,Z 955.910,A 0.000,B 0.000,C 90.000,E1 343.850} C_DIS
LIN {X -0.077,Y -176.309,Z 955.891,A 0.000,B 0.000,C 90.000,E1 340.423} C_DIS
LIN {X 0.064,Y -180.886,Z 955.872,A 0.000,B 0.000,C 90.000,E1 336.975} C_DIS
LIN {X -0.040,Y -186.181,Z 955.854,A 0.000,B 0.000,C 90.000,E1 333.640} C_DIS
LIN {X -0.106,Y -192.139,Z 955.835,A 0.000,B 0.000,C 90.000,E1 330.333} C_DIS
LIN {X -0.070,Y -198.746,Z 955.817,A 0.000,B 0.000,C 90.000,E1 327.041} C_DIS
LIN {X 0.019,Y -205.952,Z 955.799,A 0.000,B 0.000,C 90.000,E1 323.783} C_DIS
LIN {X 0.072,Y -214.649,Z 955.779,A 0.000,B 0.000,C 90.000,E1 320.194} C_DIS
LIN {X 0.044,Y -224.232,Z 955.760,A 0.000,B 0.000,C 90.000,E1 316.701} C_DIS
LIN {X -0.005,Y -233.736,Z 955.743,A 0.000,B 0.000,C 90.000,E1 313.662} C_DIS
LIN {X -0.129,Y -244.641,Z 955.726,A 0.000,B 0.000,C 90.000,E1 310.701} C_DIS
LIN {X 0.027,Y -252.237,Z 955.716,A 0.000,B 0.000,C 90.000,E1 308.830} C_DIS
LIN {X -0.011,Y -260.680,Z 955.706,A 0.000,B 0.000,C 90.000,E1 307.030} C_DIS
LIN {X 0.002,Y -271.750,Z 955.694,A 0.000,B 0.000,C 90.000,E1 304.898} C_DIS
LIN {X -0.044,Y -289.833,Z 955.677,A 0.000,B 0.000,C 90.000,E1 301.799} C_DIS
LIN {X -0.067,Y -307.171,Z 955.662,A 0.000,B 0.000,C 90.000,E1 299.127} C_DIS
LIN {X -0.176,Y -323.798,Z 955.649,A 0.000,B 0.000,C 90.000,E1 296.873} C_DIS
LIN {X 0.031,Y -344.645,Z 955.635,A 0.000,B 0.000,C 90.000,E1 294.387} C_DIS
LIN {X 0.076,Y -363.318,Z 955.624,A 0.000,B 0.000,C 90.000,E1 292.386} C_DIS
LIN {X -0.120,Y -379.462,Z 955.615,A 0.000,B 0.000,C 90.000,E1 290.791} C_DIS
LIN {X 0.155,Y -392.562,Z 955.608,A 0.000,B 0.000,C 90.000,E1 289.450} C_DIS
LIN {X 0.036,Y -403.040,Z 955.602,A 0.000,B 0.000,C 90.000,E1 288.417} C_DIS
LIN {X -0.009,Y -415.781,Z 955.595,A 0.000,B 0.000,C 90.000,E1 287.094} C_DIS
LIN {X 0.181,Y -423.277,Z 955.590,A 0.000,B 0.000,C 90.000,E1 286.260} C_DIS
LIN {X 0.101,Y -432.714,Z 955.584,A 0.000,B 0.000,C 90.000,E1 285.190} C_DIS
LIN {X 0.123,Y -441.559,Z 955.579,A 0.000,B 0.000,C 90.000,E1 284.120} C_DIS
LIN {X -0.055,Y -451.933,Z 955.571,A 0.000,B 0.000,C 90.000,E1 282.827} C_DIS
LIN {X -0.091,Y -461.885,Z 955.564,A 0.000,B 0.000,C 90.000,E1 281.535} C_DIS
LIN {X 0.080,Y -469.368,Z 955.558,A 0.000,B 0.000,C 90.000,E1 280.489} C_DIS
LIN {X 0.102,Y -474.436,Z 955.554,A 0.000,B 0.000,C 90.000,E1 279.726} C_DIS
LIN {X 0.081,Y -478.995,Z 955.550,A 0.000,B 0.000,C 90.000,E1 278.973} C_DIS
LIN {X 0.103,Y -482.797,Z 955.546,A 0.000,B 0.000,C 90.000,E1 278.219} C_DIS
LIN {X 0.093,Y -485.938,Z 955.542,A 0.000,B 0.000,C 90.000,E1 277.473} C_DIS
LIN {X -0.143,Y -487.620,Z 955.539,A 0.000,B 0.000,C 90.000,E1 277.004} C_DIS
LIN {X 0.054,Y -488.994,Z 955.536,A 0.000,B 0.000,C 90.000,E1 276.486} C_DIS
LIN {X 0.263,Y -490.046,Z 955.533,A 0.000,B 0.000,C 90.000,E1 275.967} C_DIS
LIN {X -0.057,Y -490.734,Z 955.531,A 0.000,B 0.000,C 90.000,E1 275.511} C_DIS
LIN {X 0.168,Y -491.082,Z 955.528,A 0.000,B 0.000,C 90.000,E1 274.992} C_DIS
LIN {X -0.096,Y -490.989,Z 955.525,A 0.000,B 0.000,C 90.000,E1 274.531} C_DIS
LIN {X 0.130,Y -490.470,Z 955.522,A 0.000,B 0.000,C 90.000,E1 274.012} C_DIS
LIN {X -0.168,Y -489.439,Z 955.520,A 0.000,B 0.000,C 90.000,E1 273.555} C_DIS
LIN {X 0.050,Y -487.869,Z 955.517,A 0.000,B 0.000,C 90.000,E1 273.037} C_DIS
LIN {X 0.236,Y -485.659,Z 955.514,A 0.000,B 0.000,C 90.000,E1 272.522} C_DIS
LIN {X -0.075,Y -482.753,Z 955.511,A 0.000,B 0.000,C 90.000,E1 272.064} C_DIS
LIN {X 0.098,Y -478.985,Z 955.509,A 0.000,B 0.000,C 90.000,E1 271.547} C_DIS
LIN {X 0.235,Y -474.217,Z 955.506,A 0.000,B 0.000,C 90.000,E1 271.031} C_DIS
LIN {X -0.030,Y -468.477,Z 955.503,A 0.000,B 0.000,C 90.000,E1 270.573} C_DIS
LIN {X 0.174,Y -462.520,Z 955.501,A 0.000,B 0.000,C 90.000,E1 270.115} C_DIS
LIN {X -0.191,Y -456.083,Z 955.499,A 0.000,B 0.000,C 90.000,E1 269.771} C_DIS
LIN {X -0.156,Y -449.232,Z 955.497,A 0.000,B 0.000,C 90.000,E1 269.427} C_DIS
LIN {X -0.142,Y -442.092,Z 955.495,A 0.000,B 0.000,C 90.000,E1 269.141} C_DIS
LIN {X -0.167,Y -434.910,Z 955.494,A 0.000,B 0.000,C 90.000,E1 268.912} C_DIS
LIN {X 0.109,Y -427.214,Z 955.493,A 0.000,B 0.000,C 90.000,E1 268.682} C_DIS
LIN {X -0.144,Y -419.190,Z 955.492,A 0.000,B 0.000,C 90.000,E1 268.568} C_DIS
LIN {X 0.065,Y -411.864,Z 955.491,A 0.000,B 0.000,C 90.000,E1 268.453} C_DIS
LIN {X 0.151,Y -404.103,Z 955.491,A 0.000,B 0.000,C 90.000,E1 268.396} C_DIS
LIN {X 0.042,Y -181.197,Z 955.491,A 0.000,B 0.000,C 90.000,E1 268.396} C_DIS
LIN {X -0.031,Y -180.862,Z 955.472,A 0.000,B 0.000,C 90.000,E1 265.008} C_DIS
LIN {X 0.023,Y -178.975,Z 955.444,A 0.000,B 0.000,C 90.000,E1 259.926} C_DIS
LIN {X 0.033,Y -177.937,Z 955.435,A 0.000,B 0.000,C 90.000,E1 258.229} C_DIS
LIN {X 0.047,Y -175.576,Z 955.411,A 0.000,B 0.000,C 90.000,E1 253.976} C_DIS
LIN {X 0.054,Y -172.303,Z 955.387,A 0.000,B 0.000,C 90.000,E1 249.699} C_DIS
LIN {X 0.031,Y -171.782,Z 955.383,A 0.000,B 0.000,C 90.000,E1 248.847} C_DIS
LIN {X 0.004,Y -168.712,Z 955.363,A 0.000,B 0.000,C 90.000,E1 245.409} C_DIS
LIN {X 0.043,Y -166.777,Z 955.349,A 0.000,B 0.000,C 90.000,E1 242.794} C_DIS
LIN {X -0.039,Y -162.757,Z 955.325,A 0.000,B 0.000,C 90.000,E1 238.456} C_DIS
LIN {X -0.062,Y -161.446,Z 955.315,A 0.000,B 0.000,C 90.000,E1 236.707} C_DIS
LIN {X -0.020,Y -157.440,Z 955.290,A 0.000,B 0.000,C 90.000,E1 232.271} C_DIS
LIN {X 0.014,Y -155.448,Z 955.276,A 0.000,B 0.000,C 90.000,E1 229.585} C_DIS
LIN {X 0.063,Y -151.767,Z 955.251,A 0.000,B 0.000,C 90.000,E1 225.081} C_DIS
LIN {X 0.074,Y -149.970,Z 955.236,A 0.000,B 0.000,C 90.000,E1 222.366} C_DIS
LIN {X -0.016,Y -146.807,Z 955.210,A 0.000,B 0.000,C 90.000,E1 217.855} C_DIS
LIN {X 0.001,Y -145.384,Z 955.195,A 0.000,B 0.000,C 90.000,E1 215.105} C_DIS
LIN {X -0.008,Y -142.443,Z 955.164,A 0.000,B 0.000,C 90.000,E1 209.589} C_DIS
LIN {X -0.025,Y -141.435,Z 955.149,A 0.000,B 0.000,C 90.000,E1 206.821} C_DIS
LIN {X 0.020,Y -139.366,Z 955.113,A 0.000,B 0.000,C 90.000,E1 200.301} C_DIS
LIN {X 0.007,Y -138.813,Z 955.097,A 0.000,B 0.000,C 90.000,E1 197.511} C_DIS
LIN {X 0.057,Y -138.351,Z 955.056,A 0.000,B 0.000,C 90.000,E1 190.018} C_DIS
LIN {X 0.033,Y -139.539,Z 955.004,A 0.000,B 0.000,C 90.000,E1 180.688} C_DIS
LIN {X -0.015,Y -141.233,Z 954.973,A 0.000,B 0.000,C 90.000,E1 175.122} C_DIS
LIN {X -0.056,Y -142.604,Z 954.957,A 0.000,B 0.000,C 90.000,E1 172.356} C_DIS
LIN {X 0.039,Y -144.912,Z 954.932,A 0.000,B 0.000,C 90.000,E1 167.701} C_DIS
LIN {X 0.031,Y -147.541,Z 954.911,A 0.000,B 0.000,C 90.000,E1 164.031} C_DIS
LIN {X 0.064,Y -150.142,Z 954.891,A 0.000,B 0.000,C 90.000,E1 160.369} C_DIS
LIN {X -0.067,Y -153.509,Z 954.871,A 0.000,B 0.000,C 90.000,E1 156.794} C_DIS
LIN {X -0.005,Y -157.874,Z 954.846,A 0.000,B 0.000,C 90.000,E1 152.281} C_DIS
LIN {X -0.050,Y -162.161,Z 954.826,A 0.000,B 0.000,C 90.000,E1 148.742} C_DIS
LIN {X 0.066,Y -166.368,Z 954.807,A 0.000,B 0.000,C 90.000,E1 145.182} C_DIS
LIN {X -0.066,Y -171.384,Z 954.787,A 0.000,B 0.000,C 90.000,E1 141.743} C_DIS
LIN {X 0.109,Y -176.295,Z 954.768,A 0.000,B 0.000,C 90.000,E1 138.243} C_DIS
LIN {X -0.023,Y -180.581,Z 954.754,A 0.000,B 0.000,C 90.000,E1 135.729} C_DIS
LIN {X -0.044,Y -185.983,Z 954.735,A 0.000,B 0.000,C 90.000,E1 132.366} C_DIS
LIN {X 0.011,Y -190.615,Z 954.721,A 0.000,B 0.000,C 90.000,E1 129.850} C_DIS
LIN {X 0.076,Y -194.694,Z 954.708,A 0.000,B 0.000,C 90.000,E1 127.443} C_DIS
LIN {X 0.081,Y -297.477,Z 954.708,A 0.000,B 0.000,C 90.000,E1 127.443} C_DIS
LIN {X 0.086,Y -300.913,Z 954.708,A 0.000,B 0.000,C 90.000,E1 127.363} C_DIS
LIN {X -0.149,Y -303.991,Z 954.707,A 0.000,B 0.000,C 90.000,E1 127.237} C_DIS
LIN {X -0.006,Y -307.620,Z 954.705,A 0.000,B 0.000,C 90.000,E1 126.870} C_DIS
LIN {X 0.195,Y -311.189,Z 954.702,A 0.000,B 0.000,C 90.000,E1 126.297} C_DIS
LIN {X -0.022,Y -312.719,Z 954.700,A 0.000,B 0.000,C 90.000,E1 126.011} C_DIS
LIN {X 0.014,Y -313.920,Z 954.698,A 0.000,B 0.000,C 90.000,E1 125.678} C_DIS
LIN {X 0.009,Y -324.393,Z 954.680,A 0.000,B 0.000,C 90.000,E1 122.467} C_DIS
LIN {X 0.081,Y -335.150,Z 954.665,A 0.000,B 0.000,C 90.000,E1 119.617} C_DIS
LIN {X -0.163,Y -347.284,Z 954.649,A 0.000,B 0.000,C 90.000,E1 116.873} C_DIS
LIN {X -0.076,Y -360.899,Z 954.634,A 0.000,B 0.000,C 90.000,E1 114.131} C_DIS
LIN {X -0.147,Y -374.344,Z 954.621,A 0.000,B 0.000,C 90.000,E1 111.770} C_DIS
LIN {X -0.156,Y -389.150,Z 954.608,A 0.000,B 0.000,C 90.000,E1 109.450} C_DIS
LIN {X -0.038,Y -405.425,Z 954.595,A 0.000,B 0.000,C 90.000,E1 107.166} C_DIS
LIN {X -0.016,Y -423.283,Z 954.583,A 0.000,B 0.000,C 90.000,E1 104.954} C_DIS
LIN {X -0.108,Y -442.742,Z 954.571,A 0.000,B 0.000,C 90.000,E1 102.827} C_DIS
LIN {X -0.052,Y -462.996,Z 954.560,A 0.000,B 0.000,C 90.000,E1 100.838} C_DIS
LIN {X -0.035,Y -468.005,Z 954.558,A 0.000,B 0.000,C 90.000,E1 100.366} C_DIS
LIN {X -0.089,Y -469.865,Z 954.556,A 0.000,B 0.000,C 90.000,E1 100.141} C_DIS
LIN {X -0.239,Y -471.407,Z 954.555,A 0.000,B 0.000,C 90.000,E1 99.905} C_DIS
LIN {X 0.076,Y -472.561,Z 954.553,A 0.000,B 0.000,C 90.000,E1 99.613} C_DIS
LIN {X 0.182,Y -473.950,Z 954.551,A 0.000,B 0.000,C 90.000,E1 99.095} C_DIS
LIN {X -0.099,Y -474.315,Z 954.548,A 0.000,B 0.000,C 90.000,E1 98.624} C_DIS
LIN {X 0.023,Y -473.718,Z 954.545,A 0.000,B 0.000,C 90.000,E1 98.106} C_DIS
LIN {X 0.150,Y -472.067,Z 954.542,A 0.000,B 0.000,C 90.000,E1 97.587} C_DIS
LIN {X 0.009,Y -470.755,Z 954.541,A 0.000,B 0.000,C 90.000,E1 97.352} C_DIS
LIN {X 0.072,Y -459.087,Z 954.531,A 0.000,B 0.000,C 90.000,E1 95.568} C_DIS
LIN {X 0.104,Y -445.880,Z 954.520,A 0.000,B 0.000,C 90.000,E1 93.498} C_DIS
LIN {X -0.048,Y -430.927,Z 954.506,A 0.000,B 0.000,C 90.000,E1 91.146} C_DIS
LIN {X 0.137,Y -412.328,Z 954.488,A 0.000,B 0.000,C 90.000,E1 87.879} C_DIS
LIN {X 0.192,Y -403.168,Z 954.479,A 0.000,B 0.000,C 90.000,E1 86.216} C_DIS
LIN {X -0.213,Y -390.881,Z 954.467,A 0.000,B 0.000,C 90.000,E1 84.033} C_DIS
LIN {X -0.048,Y -381.494,Z 954.457,A 0.000,B 0.000,C 90.000,E1 82.299} C_DIS
LIN {X 0.004,Y -371.878,Z 954.448,A 0.000,B 0.000,C 90.000,E1 80.557} C_DIS
LIN {X -0.117,Y -361.965,Z 954.438,A 0.000,B 0.000,C 90.000,E1 78.814} C_DIS
LIN {X 0.076,Y -351.845,Z 954.428,A 0.000,B 0.000,C 90.000,E1 76.992} C_DIS
LIN {X 0.085,Y -333.776,Z 954.409,A 0.000,B 0.000,C 90.000,E1 73.630} C_DIS
LIN {X 0.185,Y -320.014,Z 954.393,A 0.000,B 0.000,C 90.000,E1 70.786} C_DIS
LIN {X -0.093,Y -309.537,Z 954.381,A 0.000,B 0.000,C 90.000,E1 68.592} C_DIS
LIN {X -0.076,Y -297.524,Z 954.366,A 0.000,B 0.000,C 90.000,E1 65.973} C_DIS
LIN {X -0.088,Y -287.152,Z 954.353,A 0.000,B 0.000,C 90.000,E1 63.640} C_DIS
LIN {X -0.072,Y -276.831,Z 954.340,A 0.000,B 0.000,C 90.000,E1 61.257} C_DIS
LIN {X -0.047,Y -263.802,Z 954.323,A 0.000,B 0.000,C 90.000,E1 58.122} C_DIS
LIN {X 0.042,Y -251.333,Z 954.305,A 0.000,B 0.000,C 90.000,E1 54.895} C_DIS
LIN {X 0.004,Y -239.859,Z 954.287,A 0.000,B 0.000,C 90.000,E1 51.618} C_DIS
LIN {X 0.062,Y -229.321,Z 954.268,A 0.000,B 0.000,C 90.000,E1 48.243} C_DIS
LIN {X 0.029,Y -220.470,Z 954.251,A 0.000,B 0.000,C 90.000,E1 45.202} C_DIS
LIN {X -0.041,Y -212.217,Z 954.234,A 0.000,B 0.000,C 90.000,E1 42.123} C_DIS
LIN {X 0.020,Y -204.553,Z 954.216,A 0.000,B 0.000,C 90.000,E1 38.955} C_DIS
LIN {X 0.112,Y -197.525,Z 954.199,A 0.000,B 0.000,C 90.000,E1 35.724} C_DIS
LIN {X 0.018,Y -191.109,Z 954.181,A 0.000,B 0.000,C 90.000,E1 32.498} C_DIS
LIN {X -0.006,Y -185.356,Z 954.162,A 0.000,B 0.000,C 90.000,E1 29.205} C_DIS
LIN {X 0.040,Y -180.280,Z 954.144,A 0.000,B 0.000,C 90.000,E1 25.848} C_DIS
LIN {X 0.055,Y -175.893,Z 954.125,A 0.000,B 0.000,C 90.000,E1 22.461} C_DIS
LIN {X -0.069,Y -172.175,Z 954.106,A 0.000,B 0.000,C 90.000,E1 19.087} C_DIS
LIN {X -0.052,Y -168.545,Z 954.082,A 0.000,B 0.000,C 90.000,E1 14.773} C_DIS
LIN {X -0.050,Y -165.583,Z 954.053,A 0.000,B 0.000,C 90.000,E1 9.557} C_DIS
LIN {X 0.014,Y -165.814,Z 953.963,A 0.000,B 0.000,C 90.000,E1 353.394} C_DIS
LIN {X -0.036,Y -168.284,Z 953.939,A 0.000,B 0.000,C 90.000,E1 349.050} C_DIS
LIN {X 0.011,Y -171.852,Z 953.915,A 0.000,B 0.000,C 90.000,E1 344.700} C_DIS
LIN {X -0.047,Y -176.555,Z 953.891,A 0.000,B 0.000,C 90.000,E1 340.423} C_DIS
LIN {X 0.030,Y -181.130,Z 953.872,A 0.000,B 0.000,C 90.000,E1 336.997} C_DIS
LIN {X 0.005,Y -186.406,Z 953.854,A 0.000,B 0.000,C 90.000,E1 333.640} C_DIS
LIN {X -0.054,Y -192.353,Z 953.835,A 0.000,B 0.000,C 90.000,E1 330.333} C_DIS
LIN {X -0.011,Y -198.978,Z 953.817,A 0.000,B 0.000,C 90.000,E1 327.041} C_DIS
LIN {X 0.085,Y -206.161,Z 953.799,A 0.000,B 0.000,C 90.000,E1 323.783} C_DIS
LIN {X -0.058,Y -213.861,Z 953.781,A 0.000,B 0.000,C 90.000,E1 320.642} C_DIS
LIN {X 0.131,Y -222.235,Z 953.764,A 0.000,B 0.000,C 90.000,E1 317.472} C_DIS
LIN {X 0.034,Y -231.472,Z 953.747,A 0.000,B 0.000,C 90.000,E1 314.433} C_DIS
LIN {X 0.011,Y -242.021,Z 953.730,A 0.000,B 0.000,C 90.000,E1 311.434} C_DIS
LIN {X 0.126,Y -250.826,Z 953.718,A 0.000,B 0.000,C 90.000,E1 309.197} C_DIS
LIN {X -0.101,Y -260.816,Z 953.706,A 0.000,B 0.000,C 90.000,E1 307.076} C_DIS
LIN {X -0.095,Y -271.849,Z 953.694,A 0.000,B 0.000,C 90.000,E1 304.945} C_DIS
LIN {X 0.093,Y -289.864,Z 953.677,A 0.000,B 0.000,C 90.000,E1 301.799} C_DIS
LIN {X -0.070,Y -307.127,Z 953.662,A 0.000,B 0.000,C 90.000,E1 299.155} C_DIS
LIN {X -0.024,Y -323.669,Z 953.649,A 0.000,B 0.000,C 90.000,E1 296.873} C_DIS
LIN {X 0.132,Y -347.304,Z 953.634,A 0.000,B 0.000,C 90.000,E1 294.079} C_DIS
LIN {X 0.002,Y -368.623,Z 953.621,A 0.000,B 0.000,C 90.000,E1 291.844} C_DIS
LIN {X 0.148,Y -382.026,Z 953.614,A 0.000,B 0.000,C 90.000,E1 290.482} C_DIS
LIN {X -0.103,Y -395.165,Z 953.607,A 0.000,B 0.000,C 90.000,E1 289.214} C_DIS
LIN {X 0.118,Y -405.548,Z 953.601,A 0.000,B 0.000,C 90.000,E1 288.127} C_DIS
LIN {X -0.122,Y -415.708,Z 953.595,A 0.000,B 0.000,C 90.000,E1 287.094} C_DIS
LIN {X 0.187,Y -423.068,Z 953.590,A 0.000,B 0.000,C 90.000,E1 286.260} C_DIS
LIN {X 0.115,Y -432.506,Z 953.584,A 0.000,B 0.000,C 90.000,E1 285.190} C_DIS
LIN {X -0.063,Y -439.199,Z 953.580,A 0.000,B 0.000,C 90.000,E1 284.411} C_DIS
LIN {X 0.151,Y -449.737,Z 953.573,A 0.000,B 0.000,C 90.000,E1 283.063} C_DIS
LIN {X -0.085,Y -461.752,Z 953.564,A 0.000,B 0.000,C 90.000,E1 281.535} C_DIS
LIN {X 0.085,Y -469.233,Z 953.558,A 0.000,B 0.000,C 90.000,E1 280.489} C_DIS
LIN {X 0.106,Y -474.320,Z 953.554,A 0.000,B 0.000,C 90.000,E1 279.726} C_DIS
LIN {X 0.083,Y -478.905,Z 953.550,A 0.000,B 0.000,C 90.000,E1 278.973} C_DIS
LIN {X 0.105,Y -482.735,Z 953.546,A 0.000,B 0.000,C 90.000,E1 278.219} C_DIS
LIN {X 0.093,Y -485.865,Z 953.542,A 0.000,B 0.000,C 90.000,E1 277.473} C_DIS
LIN {X -0.142,Y -487.568,Z 953.539,A 0.000,B 0.000,C 90.000,E1 277.004} C_DIS
LIN {X 0.055,Y -488.963,Z 953.536,A 0.000,B 0.000,C 90.000,E1 276.486} C_DIS
LIN {X 0.263,Y -490.021,Z 953.533,A 0.000,B 0.000,C 90.000,E1 275.967} C_DIS
LIN {X -0.057,Y -490.749,Z 953.531,A 0.000,B 0.000,C 90.000,E1 275.511} C_DIS
LIN {X 0.167,Y -491.132,Z 953.528,A 0.000,B 0.000,C 90.000,E1 274.992} C_DIS
LIN {X -0.095,Y -491.059,Z 953.525,A 0.000,B 0.000,C 90.000,E1 274.531} C_DIS
LIN {X 0.130,Y -490.556,Z 953.522,A 0.000,B 0.000,C 90.000,E1 274.012} C_DIS
LIN {X -0.167,Y -489.533,Z 953.520,A 0.000,B 0.000,C 90.000,E1 273.555} C_DIS
LIN {X 0.052,Y -487.991,Z 953.517,A 0.000,B 0.000,C 90.000,E1 273.037} C_DIS
LIN {X 0.238,Y -485.748,Z 953.514,A 0.000,B 0.000,C 90.000,E1 272.522} C_DIS
LIN {X 0.082,Y -484.415,Z 953.513,A 0.000,B 0.000,C 90.000,E1 272.293} C_DIS
LIN {X -0.218,Y -481.104,Z 953.510,A 0.000,B 0.000,C 90.000,E1 271.833} C_DIS
LIN {X -0.069,Y -476.891,Z 953.507,A 0.000,B 0.000,C 90.000,E1 271.318} C_DIS
LIN {X 0.121,Y -471.704,Z 953.505,A 0.000,B 0.000,C 90.000,E1 270.802} C_DIS
LIN {X 0.095,Y -465.836,Z 953.502,A 0.000,B 0.000,C 90.000,E1 270.344} C_DIS
LIN {X 0.030,Y -459.694,Z 953.500,A 0.000,B 0.000,C 90.000,E1 269.943} C_DIS
LIN {X -0.123,Y -456.541,Z 953.499,A 0.000,B 0.000,C 90.000,E1 269.771} C_DIS
LIN {X -0.160,Y -449.584,Z 953.497,A 0.000,B 0.000,C 90.000,E1 269.427} C_DIS
LIN {X -0.184,Y -442.449,Z 953.495,A 0.000,B 0.000,C 90.000,E1 269.141} C_DIS
LIN {X 0.205,Y -435.202,Z 953.494,A 0.000,B 0.000,C 90.000,E1 268.854} C_DIS
LIN {X 0.043,Y -427.616,Z 953.493,A 0.000,B 0.000,C 90.000,E1 268.682} C_DIS
LIN {X 0.193,Y -419.728,Z 953.492,A 0.000,B 0.000,C 90.000,E1 268.511} C_DIS
LIN {X 0.190,Y -409.208,Z 953.491,A 0.000,B 0.000,C 90.000,E1 268.396} C_DIS
LIN {X -0.004,Y -403.785,Z 953.491,A 0.000,B 0.000,C 90.000,E1 268.396} C_DIS
LIN {X -0.031,Y -181.192,Z 953.491,A 0.000,B 0.000,C 90.000,E1 268.396} C_DIS
LIN {X 0.092,Y -180.857,Z 953.472,A 0.000,B 0.000,C 90.000,E1 264.951} C_DIS
LIN {X -0.034,Y -178.969,Z 953.444,A 0.000,B 0.000,C 90.000,E1 259.926} C_DIS
LIN {X -0.024,Y -177.924,Z 953.435,A 0.000,B 0.000,C 90.000,E1 258.229} C_DIS
LIN {X -0.009,Y -175.562,Z 953.411,A 0.000,B 0.000,C 90.000,E1 253.976} C_DIS
LIN {X -0.002,Y -172.291,Z 953.387,A 0.000,B 0.000,C 90.000,E1 249.699} C_DIS
LIN {X -0.024,Y -171.770,Z 953.382,A 0.000,B 0.000,C 90.000,E1 248.847} C_DIS
LIN {X -0.032,Y -168.011,Z 953.358,A 0.000,B 0.000,C 90.000,E1 244.537} C_DIS
LIN {X -0.013,Y -166.762,Z 953.349,A 0.000,B 0.000,C 90.000,E1 242.794} C_DIS
LIN {X 0.047,Y -162.741,Z 953.325,A 0.000,B 0.000,C 90.000,E1 238.408} C_DIS
LIN {X 0.108,Y -161.432,Z 953.315,A 0.000,B 0.000,C 90.000,E1 236.628} C_DIS
LIN {X -0.073,Y -157.425,Z 953.290,A 0.000,B 0.000,C 90.000,E1 232.271} C_DIS
LIN {X 0.080,Y -155.430,Z 953.275,A 0.000,B 0.000,C 90.000,E1 229.542} C_DIS
LIN {X 0.011,Y -151.753,Z 953.250,A 0.000,B 0.000,C 90.000,E1 225.081} C_DIS
LIN {X 0.023,Y -149.953,Z 953.235,A 0.000,B 0.000,C 90.000,E1 222.366} C_DIS
LIN {X 0.050,Y -146.796,Z 953.210,A 0.000,B 0.000,C 90.000,E1 217.810} C_DIS
LIN {X -0.050,Y -145.371,Z 953.195,A 0.000,B 0.000,C 90.000,E1 215.105} C_DIS
LIN {X 0.066,Y -142.435,Z 953.164,A 0.000,B 0.000,C 90.000,E1 209.539} C_DIS
LIN {X -0.011,Y -141.425,Z 953.149,A 0.000,B 0.000,C 90.000,E1 206.796} C_DIS
LIN {X -0.029,Y -139.363,Z 953.113,A 0.000,B 0.000,C 90.000,E1 200.301} C_DIS
LIN {X -0.042,Y -138.808,Z 953.097,A 0.000,B 0.000,C 90.000,E1 197.511} C_DIS
LIN {X 0.008,Y -138.351,Z 953.056,A 0.000,B 0.000,C 90.000,E1 190.018} C_DIS
LIN {X -0.016,Y -139.543,Z 953.004,A 0.000,B 0.000,C 90.000,E1 180.688} C_DIS
LIN {X -0.064,Y -141.241,Z 952.973,A 0.000,B 0.000,C 90.000,E1 175.122} C_DIS
LIN {X 0.036,Y -142.611,Z 952.957,A 0.000,B 0.000,C 90.000,E1 172.299} C_DIS
LIN {X -0.012,Y -144.925,Z 952.932,A 0.000,B 0.000,C 90.000,E1 167.701} C_DIS
LIN {X -0.019,Y -147.553,Z 952.911,A 0.000,B 0.000,C 90.000,E1 164.031} C_DIS
LIN {X 0.012,Y -150.158,Z 952.891,A 0.000,B 0.000,C 90.000,E1 160.369} C_DIS
LIN {X 0.022,Y -153.529,Z 952.871,A 0.000,B 0.000,C 90.000,E1 156.741} C_DIS
LIN {X 0.074,Y -156.947,Z 952.851,A 0.000,B 0.000,C 90.000,E1 153.127} C_DIS
LIN {X 0.011,Y -161.052,Z 952.831,A 0.000,B 0.000,C 90.000,E1 149.587} C_DIS
LIN {X 0.096,Y -163.161,Z 952.821,A 0.000,B 0.000,C 90.000,E1 147.788} C_DIS
LIN {X -0.034,Y -167.578,Z 952.802,A 0.000,B 0.000,C 90.000,E1 144.322} C_DIS
LIN {X 0.012,Y -171.408,Z 952.787,A 0.000,B 0.000,C 90.000,E1 141.698} C_DIS
LIN {X 0.051,Y -176.324,Z 952.768,A 0.000,B 0.000,C 90.000,E1 138.243} C_DIS
LIN {X -0.080,Y -180.613,Z 952.754,A 0.000,B 0.000,C 90.000,E1 135.729} C_DIS
LIN {X 0.035,Y -186.015,Z 952.735,A 0.000,B 0.000,C 90.000,E1 132.324} C_DIS
LIN {X -0.048,Y -190.649,Z 952.721,A 0.000,B 0.000,C 90.000,E1 129.850} C_DIS
LIN {X -0.085,Y -194.635,Z 952.708,A 0.000,B 0.000,C 90.000,E1 127.523} C_DIS
LIN {X -0.165,Y -297.427,Z 952.708,A 0.000,B 0.000,C 90.000,E1 127.523} C_DIS
LIN {X -0.008,Y -301.922,Z 952.708,A 0.000,B 0.000,C 90.000,E1 127.363} C_DIS
LIN {X 0.106,Y -304.728,Z 952.707,A 0.000,B 0.000,C 90.000,E1 127.156} C_DIS
LIN {X -0.062,Y -308.480,Z 952.704,A 0.000,B 0.000,C 90.000,E1 126.790} C_DIS
LIN {X -0.109,Y -310.418,Z 952.703,A 0.000,B 0.000,C 90.000,E1 126.503} C_DIS
LIN {X 0.095,Y -311.945,Z 952.701,A 0.000,B 0.000,C 90.000,E1 126.171} C_DIS
LIN {X -0.114,Y -313.282,Z 952.699,A 0.000,B 0.000,C 90.000,E1 125.884} C_DIS
LIN {X 0.038,Y -326.000,Z 952.678,A 0.000,B 0.000,C 90.000,E1 122.005} C_DIS
LIN {X -0.135,Y -336.972,Z 952.662,A 0.000,B 0.000,C 90.000,E1 119.205} C_DIS
LIN {X -0.030,Y -349.333,Z 952.647,A 0.000,B 0.000,C 90.000,E1 116.411} C_DIS
LIN {X -0.040,Y -363.198,Z 952.632,A 0.000,B 0.000,C 90.000,E1 113.695} C_DIS
LIN {X -0.052,Y -376.880,Z 952.618,A 0.000,B 0.000,C 90.000,E1 111.334} C_DIS
LIN {X -0.126,Y -391.943,Z 952.606,A 0.000,B 0.000,C 90.000,E1 109.033} C_DIS
LIN {X 0.188,Y -408.493,Z 952.593,A 0.000,B 0.000,C 90.000,E1 106.732} C_DIS
LIN {X 0.172,Y -426.651,Z 952.581,A 0.000,B 0.000,C 90.000,E1 104.537} C_DIS
LIN {X 0.243,Y -446.335,Z 952.569,A 0.000,B 0.000,C 90.000,E1 102.411} C_DIS
LIN {X 0.011,Y -466.689,Z 952.558,A 0.000,B 0.000,C 90.000,E1 100.489} C_DIS
LIN {X 0.021,Y -468.896,Z 952.557,A 0.000,B 0.000,C 90.000,E1 100.254} C_DIS
LIN {X 0.030,Y -470.561,Z 952.556,A 0.000,B 0.000,C 90.000,E1 100.018} C_DIS
LIN {X -0.118,Y -471.929,Z 952.554,A 0.000,B 0.000,C 90.000,E1 99.782} C_DIS
LIN {X 0.120,Y -472.944,Z 952.553,A 0.000,B 0.000,C 90.000,E1 99.500} C_DIS
LIN {X -0.163,Y -474.108,Z 952.550,A 0.000,B 0.000,C 90.000,E1 99.029} C_DIS
LIN {X -0.047,Y -474.275,Z 952.547,A 0.000,B 0.000,C 90.000,E1 98.511} C_DIS
LIN {X 0.078,Y -473.473,Z 952.544,A 0.000,B 0.000,C 90.000,E1 97.992} C_DIS
LIN {X 0.206,Y -471.575,Z 952.542,A 0.000,B 0.000,C 90.000,E1 97.473} C_DIS
LIN {X -0.080,Y -468.437,Z 952.539,A 0.000,B 0.000,C 90.000,E1 97.004} C_DIS
LIN {X -0.036,Y -453.464,Z 952.526,A 0.000,B 0.000,C 90.000,E1 94.702} C_DIS
LIN {X -0.118,Y -443.582,Z 952.517,A 0.000,B 0.000,C 90.000,E1 93.154} C_DIS
LIN {X -0.034,Y -425.568,Z 952.501,A 0.000,B 0.000,C 90.000,E1 90.229} C_DIS
LIN {X -0.191,Y -410.254,Z 952.486,A 0.000,B 0.000,C 90.000,E1 87.535} C_DIS
LIN {X -0.143,Y -401.030,Z 952.477,A 0.000,B 0.000,C 90.000,E1 85.869} C_DIS
LIN {X 0.184,Y -390.258,Z 952.466,A 0.000,B 0.000,C 90.000,E1 83.856} C_DIS
LIN {X -0.064,Y -379.274,Z 952.455,A 0.000,B 0.000,C 90.000,E1 81.894} C_DIS
LIN {X -0.052,Y -369.597,Z 952.445,A 0.000,B 0.000,C 90.000,E1 80.151} C_DIS
LIN {X 0.209,Y -359.627,Z 952.435,A 0.000,B 0.000,C 90.000,E1 78.342} C_DIS
LIN {X -0.069,Y -349.473,Z 952.425,A 0.000,B 0.000,C 90.000,E1 76.589} C_DIS
LIN {X 0.040,Y -331.562,Z 952.407,A 0.000,B 0.000,C 90.000,E1 73.196} C_DIS
LIN {X -0.008,Y -317.906,Z 952.391,A 0.000,B 0.000,C 90.000,E1 70.369} C_DIS
LIN {X 0.066,Y -307.434,Z 952.378,A 0.000,B 0.000,C 90.000,E1 68.103} C_DIS
LIN {X 0.021,Y -295.426,Z 952.364,A 0.000,B 0.000,C 90.000,E1 65.485} C_DIS
LIN {X -0.149,Y -286.549,Z 952.353,A 0.000,B 0.000,C 90.000,E1 63.512} C_DIS
LIN {X -0.012,Y -276.220,Z 952.339,A 0.000,B 0.000,C 90.000,E1 61.101} C_DIS
LIN {X -0.135,Y -263.197,Z 952.322,A 0.000,B 0.000,C 90.000,E1 57.995} C_DIS
LIN {X -0.063,Y -250.745,Z 952.304,A 0.000,B 0.000,C 90.000,E1 54.769} C_DIS
LIN {X 0.032,Y -239.346,Z 952.286,A 0.000,B 0.000,C 90.000,E1 51.457} C_DIS
LIN {X 0.079,Y -228.851,Z 952.267,A 0.000,B 0.000,C 90.000,E1 48.081} C_DIS
LIN {X -0.115,Y -220.052,Z 952.250,A 0.000,B 0.000,C 90.000,E1 45.081} C_DIS
LIN {X 0.118,Y -211.845,Z 952.233,A 0.000,B 0.000,C 90.000,E1 41.919} C_DIS
LIN {X -0.119,Y -204.262,Z 952.216,A 0.000,B 0.000,C 90.000,E1 38.830} C_DIS
LIN {X -0.025,Y -197.281,Z 952.198,A 0.000,B 0.000,C 90.000,E1 35.598} C_DIS
LIN {X -0.014,Y -190.928,Z 952.180,A 0.000,B 0.000,C 90.000,E1 32.339} C_DIS
LIN {X 0.022,Y -185.223,Z 952.161,A 0.000,B 0.000,C 90.000,E1 29.027} C_DIS
LIN {X -0.092,Y -180.177,Z 952.143,A 0.000,B 0.000,C 90.000,E1 25.720} C_DIS
LIN {X -0.077,Y -175.827,Z 952.124,A 0.000,B 0.000,C 90.000,E1 22.333} C_DIS
LIN {X -0.039,Y -172.161,Z 952.105,A 0.000,B 0.000,C 90.000,E1 18.906} C_DIS
LIN {X -0.024,Y -168.577,Z 952.081,A 0.000,B 0.000,C 90.000,E1 14.592} C_DIS
LIN {X -0.026,Y -165.685,Z 952.052,A 0.000,B 0.000,C 90.000,E1 9.378} C_DIS
LIN {X 0.044,Y -165.645,Z 951.968,A 0.000,B 0.000,C 90.000,E1 354.261} C_DIS
LIN {X -0.022,Y -168.511,Z 951.939,A 0.000,B 0.000,C 90.000,E1 349.050} C_DIS
LIN {X 0.033,Y -172.098,Z 951.915,A 0.000,B 0.000,C 90.000,E1 344.700} C_DIS
LIN {X -0.008,Y -175.774,Z 951.896,A 0.000,B 0.000,C 90.000,E1 341.275} C_DIS
LIN {X 0.055,Y -180.152,Z 951.877,A 0.000,B 0.000,C 90.000,E1 337.847} C_DIS
LIN {X 0.023,Y -185.249,Z 951.858,A 0.000,B 0.000,C 90.000,E1 334.485} C_DIS
LIN {X -0.068,Y -191.042,Z 951.840,A 0.000,B 0.000,C 90.000,E1 331.179} C_DIS
LIN {X 0.009,Y -197.500,Z 951.821,A 0.000,B 0.000,C 90.000,E1 327.867} C_DIS
LIN {X 0.068,Y -204.531,Z 951.803,A 0.000,B 0.000,C 90.000,E1 324.609} C_DIS
LIN {X -0.013,Y -213.087,Z 951.784,A 0.000,B 0.000,C 90.000,E1 321.045} C_DIS
LIN {X -0.016,Y -221.366,Z 951.766,A 0.000,B 0.000,C 90.000,E1 317.919} C_DIS
LIN {X 0.026,Y -230.499,Z 951.749,A 0.000,B 0.000,C 90.000,E1 314.838} C_DIS
LIN {X -0.020,Y -240.850,Z 951.732,A 0.000,B 0.000,C 90.000,E1 311.838} C_DIS
LIN {X -0.115,Y -251.016,Z 951.718,A 0.000,B 0.000,C 90.000,E1 309.277} C_DIS
LIN {X 0.019,Y -260.948,Z 951.706,A 0.000,B 0.000,C 90.000,E1 307.076} C_DIS
LIN {X -0.046,Y -273.873,Z 951.692,A 0.000,B 0.000,C 90.000,E1 304.612} C_DIS
LIN {X -0.044,Y -291.978,Z 951.675,A 0.000,B 0.000,C 90.000,E1 301.514} C_DIS
LIN {X 0.076,Y -307.080,Z 951.662,A 0.000,B 0.000,C 90.000,E1 299.155} C_DIS
LIN {X 0.129,Y -323.532,Z 951.649,A 0.000,B 0.000,C 90.000,E1 296.873} C_DIS
LIN {X 0.219,Y -344.396,Z 951.636,A 0.000,B 0.000,C 90.000,E1 294.387} C_DIS
LIN {X 0.120,Y -363.110,Z 951.624,A 0.000,B 0.000,C 90.000,E1 292.386} C_DIS
LIN {X -0.098,Y -379.204,Z 951.615,A 0.000,B 0.000,C 90.000,E1 290.791} C_DIS
LIN {X -0.043,Y -392.574,Z 951.608,A 0.000,B 0.000,C 90.000,E1 289.450} C_DIS
LIN {X -0.162,Y -402.934,Z 951.602,A 0.000,B 0.000,C 90.000,E1 288.417} C_DIS
LIN {X 0.008,Y -413.137,Z 951.596,A 0.000,B 0.000,C 90.000,E1 287.330} C_DIS
LIN {X -0.054,Y -423.128,Z 951.590,A 0.000,B 0.000,C 90.000,E1 286.260} C_DIS
LIN {X 0.104,Y -430.294,Z 951.586,A 0.000,B 0.000,C 90.000,E1 285.426} C_DIS
LIN {X -0.099,Y -437.119,Z 951.581,A 0.000,B 0.000,C 90.000,E1 284.647} C_DIS
LIN {X 0.086,Y -447.774,Z 951.574,A 0.000,B 0.000,C 90.000,E1 283.300} C_DIS
LIN {X -0.005,Y -457.940,Z 951.567,A 0.000,B 0.000,C 90.000,E1 282.007} C_DIS
LIN {X 0.209,Y -465.675,Z 951.561,A 0.000,B 0.000,C 90.000,E1 280.950} C_DIS
LIN {X 0.118,Y -471.107,Z 951.557,A 0.000,B 0.000,C 90.000,E1 280.197} C_DIS
LIN {X 0.070,Y -476.038,Z 951.552,A 0.000,B 0.000,C 90.000,E1 279.443} C_DIS
LIN {X -0.201,Y -478.994,Z 951.550,A 0.000,B 0.000,C 90.000,E1 278.973} C_DIS
LIN {X -0.180,Y -482.832,Z 951.546,A 0.000,B 0.000,C 90.000,E1 278.219} C_DIS
LIN {X -0.129,Y -485.944,Z 951.541,A 0.000,B 0.000,C 90.000,E1 277.466} C_DIS
LIN {X 0.056,Y -487.636,Z 951.539,A 0.000,B 0.000,C 90.000,E1 276.947} C_DIS
LIN {X 0.255,Y -489.035,Z 951.536,A 0.000,B 0.000,C 90.000,E1 276.429} C_DIS
LIN {X -0.024,Y -490.090,Z 951.533,A 0.000,B 0.000,C 90.000,E1 275.967} C_DIS
LIN {X 0.145,Y -490.805,Z 951.530,A 0.000,B 0.000,C 90.000,E1 275.454} C_DIS
LIN {X -0.120,Y -491.165,Z 951.528,A 0.000,B 0.000,C 90.000,E1 274.992} C_DIS
LIN {X 0.108,Y -491.093,Z 951.525,A 0.000,B 0.000,C 90.000,E1 274.473} C_DIS
LIN {X -0.156,Y -490.573,Z 951.522,A 0.000,B 0.000,C 90.000,E1 274.012} C_DIS
LIN {X 0.037,Y -489.529,Z 951.519,A 0.000,B 0.000,C 90.000,E1 273.498} C_DIS
LIN {X -0.232,Y -487.926,Z 951.517,A 0.000,B 0.000,C 90.000,E1 273.037} C_DIS
LIN {X -0.045,Y -485.691,Z 951.514,A 0.000,B 0.000,C 90.000,E1 272.522} C_DIS
LIN {X 0.128,Y -482.757,Z 951.511,A 0.000,B 0.000,C 90.000,E1 272.007} C_DIS
LIN {X -0.018,Y -480.993,Z 951.510,A 0.000,B 0.000,C 90.000,E1 271.776} C_DIS
LIN {X 0.129,Y -476.709,Z 951.507,A 0.000,B 0.000,C 90.000,E1 271.260} C_DIS
LIN {X -0.177,Y -471.461,Z 951.504,A 0.000,B 0.000,C 90.000,E1 270.802} C_DIS
LIN {X -0.204,Y -465.530,Z 951.502,A 0.000,B 0.000,C 90.000,E1 270.344} C_DIS
LIN {X 0.161,Y -459.344,Z 951.499,A 0.000,B 0.000,C 90.000,E1 269.885} C_DIS
LIN {X -0.015,Y -452.707,Z 951.497,A 0.000,B 0.000,C 90.000,E1 269.542} C_DIS
LIN {X -0.203,Y -445.775,Z 951.496,A 0.000,B 0.000,C 90.000,E1 269.255} C_DIS
LIN {X 0.000,Y -438.622,Z 951.494,A 0.000,B 0.000,C 90.000,E1 268.969} C_DIS
LIN {X 0.117,Y -431.200,Z 951.493,A 0.000,B 0.000,C 90.000,E1 268.740} C_DIS
LIN {X 0.127,Y -423.687,Z 951.492,A 0.000,B 0.000,C 90.000,E1 268.568} C_DIS
LIN {X 0.000,Y -415.130,Z 951.491,A 0.000,B 0.000,C 90.000,E1 268.453} C_DIS
LIN {X -0.121,Y -405.133,Z 951.491,A 0.000,B 0.000,C 90.000,E1 268.396} C_DIS
LIN {X -0.083,Y -181.189,Z 951.491,A 0.000,B 0.000,C 90.000,E1 268.396} C_DIS
LIN {X 0.011,Y -180.851,Z 951.472,A 0.000,B 0.000,C 90.000,E1 264.951} C_DIS
LIN {X 0.093,Y -178.961,Z 951.444,A 0.000,B 0.000,C 90.000,E1 259.859} C_DIS
LIN {X -0.015,Y -177.368,Z 951.430,A 0.000,B 0.000,C 90.000,E1 257.353} C_DIS
LIN {X 0.080,Y -175.542,Z 951.411,A 0.000,B 0.000,C 90.000,E1 253.921} C_DIS
LIN {X -0.081,Y -172.275,Z 951.387,A 0.000,B 0.000,C 90.000,E1 249.699} C_DIS
LIN {X -0.041,Y -171.754,Z 951.382,A 0.000,B 0.000,C 90.000,E1 248.827} C_DIS
LIN {X -0.024,Y -167.353,Z 951.354,A 0.000,B 0.000,C 90.000,E1 243.640} C_DIS
LIN {X 0.059,Y -166.741,Z 951.349,A 0.000,B 0.000,C 90.000,E1 242.743} C_DIS
LIN {X -0.029,Y -162.720,Z 951.324,A 0.000,B 0.000,C 90.000,E1 238.408} C_DIS
LIN {X 0.031,Y -161.411,Z 951.315,A 0.000,B 0.000,C 90.000,E1 236.628} C_DIS
LIN {X 0.073,Y -157.404,Z 951.290,A 0.000,B 0.000,C 90.000,E1 232.190} C_DIS
LIN {X 0.006,Y -155.404,Z 951.275,A 0.000,B 0.000,C 90.000,E1 229.542} C_DIS
LIN {X -0.062,Y -151.734,Z 951.250,A 0.000,B 0.000,C 90.000,E1 225.081} C_DIS
LIN {X -0.050,Y -149.930,Z 951.235,A 0.000,B 0.000,C 90.000,E1 222.366} C_DIS
LIN {X -0.022,Y -146.780,Z 951.210,A 0.000,B 0.000,C 90.000,E1 217.810} C_DIS
LIN {X 0.082,Y -145.352,Z 951.195,A 0.000,B 0.000,C 90.000,E1 215.025} C_DIS
LIN {X -0.004,Y -142.424,Z 951.164,A 0.000,B 0.000,C 90.000,E1 209.539} C_DIS
LIN {X 0.046,Y -141.412,Z 951.149,A 0.000,B 0.000,C 90.000,E1 206.744} C_DIS
LIN {X 0.032,Y -139.359,Z 951.113,A 0.000,B 0.000,C 90.000,E1 200.248} C_DIS
LIN {X 0.021,Y -138.801,Z 951.097,A 0.000,B 0.000,C 90.000,E1 197.457} C_DIS
LIN {X -0.061,Y -138.349,Z 951.056,A 0.000,B 0.000,C 90.000,E1 190.018} C_DIS
LIN {X -0.046,Y -139.367,Z 951.009,A 0.000,B 0.000,C 90.000,E1 181.604} C_DIS
LIN {X 0.006,Y -141.254,Z 950.973,A 0.000,B 0.000,C 90.000,E1 175.065} C_DIS
LIN {X -0.035,Y -142.622,Z 950.957,A 0.000,B 0.000,C 90.000,E1 172.299} C_DIS
LIN {X 0.058,Y -144.942,Z 950.932,A 0.000,B 0.000,C 90.000,E1 167.645} C_DIS
LIN {X 0.051,Y -147.571,Z 950.911,A 0.000,B 0.000,C 90.000,E1 163.976} C_DIS
LIN {X -0.060,Y -150.181,Z 950.891,A 0.000,B 0.000,C 90.000,E1 160.369} C_DIS
LIN {X -0.053,Y -153.558,Z 950.871,A 0.000,B 0.000,C 90.000,E1 156.741} C_DIS
LIN {X -0.001,Y -156.976,Z 950.851,A 0.000,B 0.000,C 90.000,E1 153.127} C_DIS
LIN {X 0.073,Y -161.086,Z 950.831,A 0.000,B 0.000,C 90.000,E1 149.537} C_DIS
LIN {X 0.018,Y -163.191,Z 950.821,A 0.000,B 0.000,C 90.000,E1 147.788} C_DIS
LIN {X 0.025,Y -167.616,Z 950.802,A 0.000,B 0.000,C 90.000,E1 144.276} C_DIS
LIN {X -0.067,Y -171.443,Z 950.787,A 0.000,B 0.000,C 90.000,E1 141.698} C_DIS
LIN {X -0.030,Y -176.365,Z 950.768,A 0.000,B 0.000,C 90.000,E1 138.243} C_DIS
LIN {X 0.093,Y -180.657,Z 950.754,A 0.000,B 0.000,C 90.000,E1 135.648} C_DIS
LIN {X 0.076,Y -186.059,Z 950.735,A 0.000,B 0.000,C 90.000,E1 132.285} C_DIS
LIN {X 0.013,Y -190.695,Z 950.721,A 0.000,B 0.000,C 90.000,E1 129.806} C_DIS
LIN {X 0.022,Y -194.577,Z 950.708,A 0.000,B 0.000,C 90.000,E1 127.523} C_DIS
LIN {X -0.001,Y -297.461,Z 950.708,A 0.000,B 0.000,C 90.000,E1 127.523} C_DIS
LIN {X 0.100,Y -302.836,Z 950.707,A 0.000,B 0.000,C 90.000,E1 127.317} C_DIS
LIN {X 0.034,Y -305.660,Z 950.706,A 0.000,B 0.000,C 90.000,E1 127.111} C_DIS
LIN {X -0.028,Y -309.427,Z 950.704,A 0.000,B 0.000,C 90.000,E1 126.664} C_DIS
LIN {X 0.192,Y -311.290,Z 950.702,A 0.000,B 0.000,C 90.000,E1 126.297} C_DIS
LIN {X -0.023,Y -312.745,Z 950.700,A 0.000,B 0.000,C 90.000,E1 126.011} C_DIS
LIN {X -0.001,Y -314.865,Z 950.696,A 0.000,B 0.000,C 90.000,E1 125.358} C_DIS
LIN {X 0.106,Y -325.476,Z 950.679,A 0.000,B 0.000,C 90.000,E1 122.133} C_DIS
LIN {X -0.078,Y -336.381,Z 950.663,A 0.000,B 0.000,C 90.000,E1 119.333} C_DIS
LIN {X 0.006,Y -348.674,Z 950.647,A 0.000,B 0.000,C 90.000,E1 116.539} C_DIS
LIN {X -0.015,Y -362.459,Z 950.632,A 0.000,B 0.000,C 90.000,E1 113.823} C_DIS
LIN {X -0.043,Y -376.067,Z 950.619,A 0.000,B 0.000,C 90.000,E1 111.461} C_DIS
LIN {X -0.006,Y -391.050,Z 950.606,A 0.000,B 0.000,C 90.000,E1 109.141} C_DIS
LIN {X 0.163,Y -407.515,Z 950.594,A 0.000,B 0.000,C 90.000,E1 106.858} C_DIS
LIN {X 0.129,Y -425.581,Z 950.582,A 0.000,B 0.000,C 90.000,E1 104.662} C_DIS
LIN {X 0.159,Y -445.192,Z 950.570,A 0.000,B 0.000,C 90.000,E1 102.535} C_DIS
LIN {X -0.051,Y -467.976,Z 950.558,A 0.000,B 0.000,C 90.000,E1 100.366} C_DIS
LIN {X -0.177,Y -469.908,Z 950.556,A 0.000,B 0.000,C 90.000,E1 100.141} C_DIS
LIN {X -0.220,Y -471.373,Z 950.555,A 0.000,B 0.000,C 90.000,E1 99.905} C_DIS
LIN {X -0.048,Y -473.383,Z 950.552,A 0.000,B 0.000,C 90.000,E1 99.378} C_DIS
LIN {X 0.058,Y -474.261,Z 950.549,A 0.000,B 0.000,C 90.000,E1 98.859} C_DIS
LIN {X 0.179,Y -474.163,Z 950.546,A 0.000,B 0.000,C 90.000,E1 98.341} C_DIS
LIN {X -0.097,Y -473.080,Z 950.544,A 0.000,B 0.000,C 90.000,E1 97.871} C_DIS
LIN {X 0.167,Y -472.119,Z 950.542,A 0.000,B 0.000,C 90.000,E1 97.587} C_DIS
LIN {X 0.027,Y -470.823,Z 950.541,A 0.000,B 0.000,C 90.000,E1 97.352} C_DIS
LIN {X -0.092,Y -457.526,Z 950.530,A 0.000,B 0.000,C 90.000,E1 95.334} C_DIS
LIN {X 0.120,Y -446.038,Z 950.520,A 0.000,B 0.000,C 90.000,E1 93.498} C_DIS
LIN {X -0.180,Y -432.797,Z 950.508,A 0.000,B 0.000,C 90.000,E1 91.432} C_DIS
LIN {X 0.073,Y -413.999,Z 950.490,A 0.000,B 0.000,C 90.000,E1 88.165} C_DIS
LIN {X 0.163,Y -404.835,Z 950.481,A 0.000,B 0.000,C 90.000,E1 86.502} C_DIS
LIN {X 0.193,Y -392.494,Z 950.468,A 0.000,B 0.000,C 90.000,E1 84.261} C_DIS
LIN {X -0.013,Y -381.592,Z 950.457,A 0.000,B 0.000,C 90.000,E1 82.299} C_DIS
LIN {X 0.040,Y -371.948,Z 950.448,A 0.000,B 0.000,C 90.000,E1 80.557} C_DIS
LIN {X -0.080,Y -362.070,Z 950.438,A 0.000,B 0.000,C 90.000,E1 78.814} C_DIS
LIN {X 0.113,Y -351.949,Z 950.428,A 0.000,B 0.000,C 90.000,E1 76.992} C_DIS
LIN {X 0.119,Y -333.809,Z 950.409,A 0.000,B 0.000,C 90.000,E1 73.630} C_DIS
LIN {X -0.184,Y -320.087,Z 950.393,A 0.000,B 0.000,C 90.000,E1 70.859} C_DIS
LIN {X 0.022,Y -311.113,Z 950.383,A 0.000,B 0.000,C 90.000,E1 68.901} C_DIS
LIN {X 0.060,Y -300.602,Z 950.370,A 0.000,B 0.000,C 90.000,E1 66.613} C_DIS
LIN {X -0.033,Y -288.713,Z 950.355,A 0.000,B 0.000,C 90.000,E1 63.973} C_DIS
LIN {X 0.011,Y -278.353,Z 950.342,A 0.000,B 0.000,C 90.000,E1 61.591} C_DIS
LIN {X -0.146,Y -268.082,Z 950.329,A 0.000,B 0.000,C 90.000,E1 59.203} C_DIS
LIN {X 0.027,Y -256.775,Z 950.313,A 0.000,B 0.000,C 90.000,E1 56.342} C_DIS
LIN {X -0.143,Y -244.826,Z 950.295,A 0.000,B 0.000,C 90.000,E1 53.130} C_DIS
LIN {X 0.089,Y -233.899,Z 950.276,A 0.000,B 0.000,C 90.000,E1 49.747} C_DIS
LIN {X -0.038,Y -223.756,Z 950.258,A 0.000,B 0.000,C 90.000,E1 46.377} C_DIS
LIN {X -0.033,Y -215.341,Z 950.240,A 0.000,B 0.000,C 90.000,E1 43.299} C_DIS
LIN {X -0.050,Y -207.532,Z 950.223,A 0.000,B 0.000,C 90.000,E1 40.172} C_DIS
LIN {X 0.088,Y -200.311,Z 950.205,A 0.000,B 0.000,C 90.000,E1 36.950} C_DIS
LIN {X 0.119,Y -193.700,Z 950.187,A 0.000,B 0.000,C 90.000,E1 33.706} C_DIS
LIN {X -0.008,Y -187.711,Z 950.169,A 0.000,B 0.000,C 90.000,E1 30.463} C_DIS
LIN {X 0.020,Y -182.422,Z 950.151,A 0.000,B 0.000,C 90.000,E1 27.129} C_DIS
LIN {X 0.000,Y -177.773,Z 950.132,A 0.000,B 0.000,C 90.000,E1 23.770} C_DIS
LIN {X -0.014,Y -173.814,Z 950.113,A 0.000,B 0.000,C 90.000,E1 20.375} C_DIS
LIN {X -0.006,Y -169.822,Z 950.089,A 0.000,B 0.000,C 90.000,E1 16.079} C_DIS
LIN {X -0.072,Y -167.006,Z 950.065,A 0.000,B 0.000,C 90.000,E1 11.771} C_DIS
LIN {X 0.040,Y -164.742,Z 950.031,A 0.000,B 0.000,C 90.000,E1 5.625} C_DIS
LIN {X 0.051,Y -165.855,Z 949.968,A 0.000,B 0.000,C 90.000,E1 354.261} C_DIS
LIN {X -0.026,Y -168.154,Z 949.944,A 0.000,B 0.000,C 90.000,E1 349.926} C_DIS
LIN {X -0.023,Y -171.524,Z 949.920,A 0.000,B 0.000,C 90.000,E1 345.589} C_DIS
LIN {X 0.021,Y -176.019,Z 949.896,A 0.000,B 0.000,C 90.000,E1 341.275} C_DIS
LIN {X 0.091,Y -180.389,Z 949.877,A 0.000,B 0.000,C 90.000,E1 337.847} C_DIS
LIN {X -0.102,Y -185.482,Z 949.858,A 0.000,B 0.000,C 90.000,E1 334.537} C_DIS
LIN {X -0.017,Y -191.282,Z 949.840,A 0.000,B 0.000,C 90.000,E1 331.179} C_DIS
LIN {X 0.067,Y -197.745,Z 949.822,A 0.000,B 0.000,C 90.000,E1 327.867} C_DIS
LIN {X 0.015,Y -204.752,Z 949.804,A 0.000,B 0.000,C 90.000,E1 324.642} C_DIS
LIN {X -0.104,Y -213.325,Z 949.784,A 0.000,B 0.000,C 90.000,E1 321.090} C_DIS
LIN {X 0.068,Y -221.586,Z 949.766,A 0.000,B 0.000,C 90.000,E1 317.919} C_DIS
LIN {X 0.120,Y -230.741,Z 949.749,A 0.000,B 0.000,C 90.000,E1 314.838} C_DIS
LIN {X 0.084,Y -241.083,Z 949.733,A 0.000,B 0.000,C 90.000,E1 311.838} C_DIS
LIN {X -0.002,Y -251.216,Z 949.718,A 0.000,B 0.000,C 90.000,E1 309.277} C_DIS
LIN {X 0.140,Y -261.092,Z 949.706,A 0.000,B 0.000,C 90.000,E1 307.076} C_DIS
LIN {X 0.084,Y -273.930,Z 949.692,A 0.000,B 0.000,C 90.000,E1 304.612} C_DIS
LIN {X -0.057,Y -291.990,Z 949.675,A 0.000,B 0.000,C 90.000,E1 301.544} C_DIS
LIN {X -0.020,Y -309.286,Z 949.660,A 0.000,B 0.000,C 90.000,E1 298.871} C_DIS
LIN {X -0.005,Y -323.389,Z 949.650,A 0.000,B 0.000,C 90.000,E1 296.924} C_DIS
LIN {X -0.034,Y -344.102,Z 949.636,A 0.000,B 0.000,C 90.000,E1 294.463} C_DIS
LIN {X -0.058,Y -360.158,Z 949.626,A 0.000,B 0.000,C 90.000,E1 292.717} C_DIS
LIN {X 0.059,Y -378.862,Z 949.616,A 0.000,B 0.000,C 90.000,E1 290.791} C_DIS
LIN {X 0.110,Y -392.221,Z 949.608,A 0.000,B 0.000,C 90.000,E1 289.450} C_DIS
LIN {X -0.058,Y -402.588,Z 949.602,A 0.000,B 0.000,C 90.000,E1 288.417} C_DIS
LIN {X 0.077,Y -412.841,Z 949.596,A 0.000,B 0.000,C 90.000,E1 287.330} C_DIS
LIN {X 0.202,Y -422.590,Z 949.591,A 0.000,B 0.000,C 90.000,E1 286.260} C_DIS
LIN {X -0.055,Y -429.837,Z 949.586,A 0.000,B 0.000,C 90.000,E1 285.481} C_DIS
LIN {X -0.075,Y -438.822,Z 949.580,A 0.000,B 0.000,C 90.000,E1 284.411} C_DIS
LIN {X 0.133,Y -449.421,Z 949.573,A 0.000,B 0.000,C 90.000,E1 283.063} C_DIS
LIN {X 0.072,Y -459.531,Z 949.565,A 0.000,B 0.000,C 90.000,E1 281.771} C_DIS
LIN {X -0.241,Y -467.180,Z 949.560,A 0.000,B 0.000,C 90.000,E1 280.782} C_DIS
LIN {X 0.220,Y -472.471,Z 949.555,A 0.000,B 0.000,C 90.000,E1 279.962} C_DIS
LIN {X 0.190,Y -477.243,Z 949.551,A 0.000,B 0.000,C 90.000,E1 279.208} C_DIS
LIN {X 0.196,Y -481.391,Z 949.547,A 0.000,B 0.000,C 90.000,E1 278.454} C_DIS
LIN {X -0.118,Y -483.754,Z 949.544,A 0.000,B 0.000,C 90.000,E1 277.992} C_DIS
LIN {X 0.060,Y -485.792,Z 949.542,A 0.000,B 0.000,C 90.000,E1 277.473} C_DIS
LIN {X -0.175,Y -487.536,Z 949.539,A 0.000,B 0.000,C 90.000,E1 277.004} C_DIS
LIN {X 0.021,Y -488.952,Z 949.536,A 0.000,B 0.000,C 90.000,E1 276.486} C_DIS
LIN {X 0.228,Y -490.050,Z 949.533,A 0.000,B 0.000,C 90.000,E1 275.967} C_DIS
LIN {X -0.091,Y -490.808,Z 949.531,A 0.000,B 0.000,C 90.000,E1 275.511} C_DIS
LIN {X 0.133,Y -491.190,Z 949.528,A 0.000,B 0.000,C 90.000,E1 274.992} C_DIS
LIN {X -0.129,Y -491.161,Z 949.525,A 0.000,B 0.000,C 90.000,E1 274.531} C_DIS
LIN {X 0.097,Y -490.697,Z 949.522,A 0.000,B 0.000,C 90.000,E1 274.012} C_DIS
LIN {X -0.200,Y -489.718,Z 949.520,A 0.000,B 0.000,C 90.000,E1 273.555} C_DIS
LIN {X 0.020,Y -488.177,Z 949.517,A 0.000,B 0.000,C 90.000,E1 273.037} C_DIS
LIN {X 0.207,Y -485.992,Z 949.514,A 0.000,B 0.000,C 90.000,E1 272.522} C_DIS
LIN {X -0.103,Y -483.099,Z 949.511,A 0.000,B 0.000,C 90.000,E1 272.064} C_DIS
LIN {X 0.073,Y -479.381,Z 949.509,A 0.000,B 0.000,C 90.000,E1 271.547} C_DIS
LIN {X 0.212,Y -474.738,Z 949.506,A 0.000,B 0.000,C 90.000,E1 271.031} C_DIS
LIN {X -0.122,Y -468.935,Z 949.503,A 0.000,B 0.000,C 90.000,E1 270.573} C_DIS
LIN {X 0.042,Y -463.028,Z 949.501,A 0.000,B 0.000,C 90.000,E1 270.115} C_DIS
LIN {X 0.072,Y -456.504,Z 949.498,A 0.000,B 0.000,C 90.000,E1 269.714} C_DIS
LIN {X 0.114,Y -449.811,Z 949.497,A 0.000,B 0.000,C 90.000,E1 269.370} C_DIS
LIN {X 0.100,Y -442.769,Z 949.495,A 0.000,B 0.000,C 90.000,E1 269.083} C_DIS
LIN {X 0.004,Y -435.487,Z 949.494,A 0.000,B 0.000,C 90.000,E1 268.854} C_DIS
LIN {X -0.177,Y -427.996,Z 949.493,A 0.000,B 0.000,C 90.000,E1 268.682} C_DIS
LIN {X -0.065,Y -420.213,Z 949.492,A 0.000,B 0.000,C 90.000,E1 268.511} C_DIS
LIN {X -0.098,Y -409.773,Z 949.491,A 0.000,B 0.000,C 90.000,E1 268.396} C_DIS
LIN {X 0.108,Y -403.854,Z 949.491,A 0.000,B 0.000,C 90.000,E1 268.339} C_DIS
LIN {X 0.018,Y -181.185,Z 949.491,A 0.000,B 0.000,C 90.000,E1 268.339} C_DIS
LIN {X -0.045,Y -180.847,Z 949.472,A 0.000,B 0.000,C 90.000,E1 264.951} C_DIS
LIN {X 0.038,Y -178.955,Z 949.444,A 0.000,B 0.000,C 90.000,E1 259.859} C_DIS
LIN {X -0.070,Y -177.357,Z 949.430,A 0.000,B 0.000,C 90.000,E1 257.353} C_DIS
LIN {X 0.025,Y -175.528,Z 949.411,A 0.000,B 0.000,C 90.000,E1 253.921} C_DIS
LIN {X 0.027,Y -172.263,Z 949.387,A 0.000,B 0.000,C 90.000,E1 249.645} C_DIS
LIN {X 0.065,Y -171.742,Z 949.382,A 0.000,B 0.000,C 90.000,E1 248.773} C_DIS
LIN {X -0.076,Y -167.340,Z 949.353,A 0.000,B 0.000,C 90.000,E1 243.640} C_DIS
LIN {X 0.006,Y -166.726,Z 949.349,A 0.000,B 0.000,C 90.000,E1 242.743} C_DIS
LIN {X -0.081,Y -162.706,Z 949.324,A 0.000,B 0.000,C 90.000,E1 238.408} C_DIS
LIN {X -0.020,Y -161.397,Z 949.315,A 0.000,B 0.000,C 90.000,E1 236.628} C_DIS
LIN {X 0.023,Y -157.390,Z 949.290,A 0.000,B 0.000,C 90.000,E1 232.190} C_DIS
LIN {X -0.044,Y -155.386,Z 949.275,A 0.000,B 0.000,C 90.000,E1 229.542} C_DIS
LIN {X -0.005,Y -151.722,Z 949.250,A 0.000,B 0.000,C 90.000,E1 225.040} C_DIS
LIN {X 0.011,Y -149.915,Z 949.235,A 0.000,B 0.000,C 90.000,E1 222.324} C_DIS
LIN {X -0.071,Y -146.770,Z 949.210,A 0.000,B 0.000,C 90.000,E1 217.810} C_DIS
LIN {X 0.034,Y -145.339,Z 949.195,A 0.000,B 0.000,C 90.000,E1 215.025} C_DIS
LIN {X -0.052,Y -142.416,Z 949.164,A 0.000,B 0.000,C 90.000,E1 209.539} C_DIS
LIN {X -0.002,Y -141.402,Z 949.149,A 0.000,B 0.000,C 90.000,E1 206.744} C_DIS
LIN {X -0.015,Y -139.356,Z 949.112,A 0.000,B 0.000,C 90.000,E1 200.248} C_DIS
LIN {X -0.027,Y -138.796,Z 949.097,A 0.000,B 0.000,C 90.000,E1 197.457} C_DIS
LIN {X 0.028,Y -138.348,Z 949.055,A 0.000,B 0.000,C 90.000,E1 189.962} C_DIS
LIN {X 0.046,Y -139.373,Z 949.009,A 0.000,B 0.000,C 90.000,E1 181.547} C_DIS
LIN {X -0.041,Y -141.263,Z 948.972,A 0.000,B 0.000,C 90.000,E1 175.065} C_DIS
LIN {X 0.059,Y -142.629,Z 948.957,A 0.000,B 0.000,C 90.000,E1 172.243} C_DIS
LIN {X 0.011,Y -144.955,Z 948.931,A 0.000,B 0.000,C 90.000,E1 167.645} C_DIS
LIN {X 0.001,Y -147.583,Z 948.911,A 0.000,B 0.000,C 90.000,E1 163.976} C_DIS
LIN {X 0.031,Y -150.196,Z 948.891,A 0.000,B 0.000,C 90.000,E1 160.315} C_DIS
LIN {X -0.042,Y -153.578,Z 948.871,A 0.000,B 0.000,C 90.000,E1 156.719} C_DIS
LIN {X -0.052,Y -156.995,Z 948.851,A 0.000,B 0.000,C 90.000,E1 153.127} C_DIS
LIN {X 0.021,Y -161.110,Z 948.831,A 0.000,B 0.000,C 90.000,E1 149.537} C_DIS
LIN {X -0.034,Y -163.212,Z 948.821,A 0.000,B 0.000,C 90.000,E1 147.788} C_DIS
LIN {X -0.029,Y -167.641,Z 948.801,A 0.000,B 0.000,C 90.000,E1 144.276} C_DIS
LIN {X -0.015,Y -171.466,Z 948.787,A 0.000,B 0.000,C 90.000,E1 141.662} C_DIS
LIN {X -0.084,Y -176.393,Z 948.768,A 0.000,B 0.000,C 90.000,E1 138.243} C_DIS
LIN {X 0.037,Y -180.686,Z 948.754,A 0.000,B 0.000,C 90.000,E1 135.648} C_DIS
LIN {X 0.020,Y -186.090,Z 948.735,A 0.000,B 0.000,C 90.000,E1 132.285} C_DIS
LIN {X -0.044,Y -190.726,Z 948.721,A 0.000,B 0.000,C 90.000,E1 129.806} C_DIS
LIN {X -0.008,Y -194.512,Z 948.709,A 0.000,B 0.000,C 90.000,E1 127.569} C_DIS
LIN {X -0.053,Y -296.947,Z 948.709,A 0.000,B 0.000,C 90.000,E1 127.569} C_DIS
LIN {X 0.062,Y -298.695,Z 948.709,A 0.000,B 0.000,C 90.000,E1 127.523} C_DIS
LIN {X 0.010,Y -303.473,Z 948.707,A 0.000,B 0.000,C 90.000,E1 127.317} C_DIS
LIN {X 0.037,Y -306.646,Z 948.706,A 0.000,B 0.000,C 90.000,E1 127.030} C_DIS
LIN {X 0.112,Y -310.323,Z 948.703,A 0.000,B 0.000,C 90.000,E1 126.503} C_DIS
LIN {X -0.108,Y -311.965,Z 948.701,A 0.000,B 0.000,C 90.000,E1 126.217} C_DIS
LIN {X -0.077,Y -313.254,Z 948.699,A 0.000,B 0.000,C 90.000,E1 125.884} C_DIS
LIN {X -0.017,Y -324.796,Z 948.680,A 0.000,B 0.000,C 90.000,E1 122.339} C_DIS
LIN {X 0.067,Y -335.617,Z 948.664,A 0.000,B 0.000,C 90.000,E1 119.489} C_DIS
LIN {X -0.159,Y -347.814,Z 948.648,A 0.000,B 0.000,C 90.000,E1 116.744} C_DIS
LIN {X -0.062,Y -361.502,Z 948.633,A 0.000,B 0.000,C 90.000,E1 114.003} C_DIS
LIN {X -0.120,Y -375.015,Z 948.620,A 0.000,B 0.000,C 90.000,E1 111.642} C_DIS
LIN {X -0.114,Y -389.896,Z 948.607,A 0.000,B 0.000,C 90.000,E1 109.322} C_DIS
LIN {X 0.020,Y -406.250,Z 948.595,A 0.000,B 0.000,C 90.000,E1 107.040} C_DIS
LIN {X 0.058,Y -424.194,Z 948.582,A 0.000,B 0.000,C 90.000,E1 104.828} C_DIS
LIN {X 0.000,Y -443.728,Z 948.571,A 0.000,B 0.000,C 90.000,E1 102.703} C_DIS
LIN {X 0.122,Y -464.011,Z 948.560,A 0.000,B 0.000,C 90.000,E1 100.715} C_DIS
LIN {X 0.054,Y -466.571,Z 948.558,A 0.000,B 0.000,C 90.000,E1 100.489} C_DIS
LIN {X 0.072,Y -468.806,Z 948.557,A 0.000,B 0.000,C 90.000,E1 100.254} C_DIS
LIN {X -0.081,Y -470.619,Z 948.556,A 0.000,B 0.000,C 90.000,E1 100.018} C_DIS
LIN {X 0.228,Y -471.981,Z 948.554,A 0.000,B 0.000,C 90.000,E1 99.726} C_DIS
LIN {X -0.139,Y -473.692,Z 948.551,A 0.000,B 0.000,C 90.000,E1 99.265} C_DIS
LIN {X -0.029,Y -474.329,Z 948.549,A 0.000,B 0.000,C 90.000,E1 98.746} C_DIS
LIN {X 0.163,Y -474.001,Z 948.546,A 0.000,B 0.000,C 90.000,E1 98.219} C_DIS
LIN {X -0.180,Y -472.663,Z 948.543,A 0.000,B 0.000,C 90.000,E1 97.757} C_DIS
LIN {X 0.086,Y -471.549,Z 948.542,A 0.000,B 0.000,C 90.000,E1 97.473} C_DIS
LIN {X -0.203,Y -468.382,Z 948.539,A 0.000,B 0.000,C 90.000,E1 97.004} C_DIS
LIN {X -0.151,Y -453.491,Z 948.526,A 0.000,B 0.000,C 90.000,E1 94.702} C_DIS
LIN {X -0.207,Y -443.654,Z 948.517,A 0.000,B 0.000,C 90.000,E1 93.151} C_DIS
LIN {X 0.005,Y -428.885,Z 948.504,A 0.000,B 0.000,C 90.000,E1 90.745} C_DIS
LIN {X 0.034,Y -411.837,Z 948.488,A 0.000,B 0.000,C 90.000,E1 87.764} C_DIS
LIN {X 0.080,Y -402.577,Z 948.478,A 0.000,B 0.000,C 90.000,E1 86.102} C_DIS
LIN {X 0.035,Y -391.785,Z 948.468,A 0.000,B 0.000,C 90.000,E1 84.147} C_DIS
LIN {X -0.184,Y -380.844,Z 948.456,A 0.000,B 0.000,C 90.000,E1 82.186} C_DIS
LIN {X -0.143,Y -371.165,Z 948.447,A 0.000,B 0.000,C 90.000,E1 80.443} C_DIS
LIN {X 0.150,Y -361.309,Z 948.437,A 0.000,B 0.000,C 90.000,E1 78.634} C_DIS
LIN {X -0.096,Y -351.145,Z 948.427,A 0.000,B 0.000,C 90.000,E1 76.881} C_DIS
LIN {X -0.021,Y -333.054,Z 948.408,A 0.000,B 0.000,C 90.000,E1 73.504} C_DIS
LIN {X -0.032,Y -319.389,Z 948.393,A 0.000,B 0.000,C 90.000,E1 70.678} C_DIS
LIN {X 0.073,Y -308.923,Z 948.380,A 0.000,B 0.000,C 90.000,E1 68.411} C_DIS
LIN {X 0.063,Y -298.427,Z 948.367,A 0.000,B 0.000,C 90.000,E1 66.125} C_DIS
LIN {X -0.077,Y -288.027,Z 948.354,A 0.000,B 0.000,C 90.000,E1 63.819} C_DIS
LIN {X -0.037,Y -277.656,Z 948.341,A 0.000,B 0.000,C 90.000,E1 61.435} C_DIS
LIN {X -0.041,Y -265.962,Z 948.326,A 0.000,B 0.000,C 90.000,E1 58.663} C_DIS
LIN {X -0.040,Y -253.338,Z 948.308,A 0.000,B 0.000,C 90.000,E1 55.468} C_DIS
LIN {X -0.017,Y -241.727,Z 948.290,A 0.000,B 0.000,C 90.000,E1 52.190} C_DIS
LIN {X -0.058,Y -231.038,Z 948.271,A 0.000,B 0.000,C 90.000,E1 48.852} C_DIS
LIN {X 0.052,Y -221.092,Z 948.252,A 0.000,B 0.000,C 90.000,E1 45.405} C_DIS
LIN {X 0.006,Y -212.896,Z 948.235,A 0.000,B 0.000,C 90.000,E1 42.324} C_DIS
LIN {X -0.066,Y -205.333,Z 948.218,A 0.000,B 0.000,C 90.000,E1 39.197} C_DIS
LIN {X 0.053,Y -198.310,Z 948.200,A 0.000,B 0.000,C 90.000,E1 35.964} C_DIS
LIN {X -0.071,Y -191.908,Z 948.182,A 0.000,B 0.000,C 90.000,E1 32.752} C_DIS
LIN {X 0.086,Y -186.170,Z 948.164,A 0.000,B 0.000,C 90.000,E1 29.411} C_DIS
LIN {X -0.008,Y -181.061,Z 948.145,A 0.000,B 0.000,C 90.000,E1 26.104} C_DIS
LIN {X 0.028,Y -176.642,Z 948.126,A 0.000,B 0.000,C 90.000,E1 22.717} C_DIS
LIN {X -0.017,Y -172.897,Z 948.107,A 0.000,B 0.000,C 90.000,E1 19.322} C_DIS
LIN {X 0.018,Y -169.210,Z 948.083,A 0.000,B 0.000,C 90.000,E1 15.009} C_DIS
LIN {X 0.044,Y -166.240,Z 948.055,A 0.000,B 0.000,C 90.000,E1 9.792} C_DIS
LIN {X -0.066,Y -164.528,Z 948.006,A 0.000,B 0.000,C 90.000,E1 1.088} C_DIS
LIN {X 0.040,Y -166.440,Z 947.963,A 0.000,B 0.000,C 90.000,E1 353.394} C_DIS
LIN {X 0.033,Y -169.579,Z 947.934,A 0.000,B 0.000,C 90.000,E1 348.173} C_DIS
LIN {X -0.089,Y -172.583,Z 947.915,A 0.000,B 0.000,C 90.000,E1 344.755} C_DIS
LIN {X 0.045,Y -177.283,Z 947.891,A 0.000,B 0.000,C 90.000,E1 340.423} C_DIS
LIN {X -0.024,Y -181.844,Z 947.872,A 0.000,B 0.000,C 90.000,E1 337.050} C_DIS
LIN {X -0.029,Y -187.099,Z 947.854,A 0.000,B 0.000,C 90.000,E1 333.691} C_DIS
LIN {X -0.067,Y -193.062,Z 947.835,A 0.000,B 0.000,C 90.000,E1 330.383} C_DIS
LIN {X -0.107,Y -199.676,Z 947.817,A 0.000,B 0.000,C 90.000,E1 327.120} C_DIS
LIN {X 0.000,Y -206.861,Z 947.799,A 0.000,B 0.000,C 90.000,E1 323.863} C_DIS
LIN {X 0.078,Y -215.560,Z 947.779,A 0.000,B 0.000,C 90.000,E1 320.275} C_DIS
LIN {X -0.002,Y -224.020,Z 947.762,A 0.000,B 0.000,C 90.000,E1 317.187} C_DIS
LIN {X 0.101,Y -233.474,Z 947.745,A 0.000,B 0.000,C 90.000,E1 314.109} C_DIS
LIN {X -0.031,Y -244.088,Z 947.729,A 0.000,B 0.000,C 90.000,E1 311.148} C_DIS
LIN {X 0.128,Y -252.973,Z 947.716,A 0.000,B 0.000,C 90.000,E1 308.910} C_DIS
LIN {X -0.102,Y -261.242,Z 947.706,A 0.000,B 0.000,C 90.000,E1 307.156} C_DIS
LIN {X -0.008,Y -273.993,Z 947.693,A 0.000,B 0.000,C 90.000,E1 304.659} C_DIS
LIN {X 0.087,Y -292.009,Z 947.675,A 0.000,B 0.000,C 90.000,E1 301.544} C_DIS
LIN {X 0.106,Y -306.989,Z 947.662,A 0.000,B 0.000,C 90.000,E1 299.205} C_DIS
LIN {X 0.086,Y -320.780,Z 947.651,A 0.000,B 0.000,C 90.000,E1 297.257} C_DIS
LIN {X 0.113,Y -338.474,Z 947.639,A 0.000,B 0.000,C 90.000,E1 295.079} C_DIS
LIN {X 0.088,Y -357.001,Z 947.628,A 0.000,B 0.000,C 90.000,E1 293.025} C_DIS
LIN {X -0.024,Y -378.306,Z 947.616,A 0.000,B 0.000,C 90.000,E1 290.844} C_DIS
LIN {X 0.021,Y -391.660,Z 947.608,A 0.000,B 0.000,C 90.000,E1 289.504} C_DIS
LIN {X -0.021,Y -404.613,Z 947.601,A 0.000,B 0.000,C 90.000,E1 288.181} C_DIS
LIN {X 0.112,Y -414.816,Z 947.595,A 0.000,B 0.000,C 90.000,E1 287.094} C_DIS
LIN {X 0.022,Y -424.726,Z 947.589,A 0.000,B 0.000,C 90.000,E1 286.024} C_DIS
LIN {X 0.188,Y -431.858,Z 947.585,A 0.000,B 0.000,C 90.000,E1 285.190} C_DIS
LIN {X 0.201,Y -440.738,Z 947.579,A 0.000,B 0.000,C 90.000,E1 284.120} C_DIS
LIN {X 0.014,Y -451.268,Z 947.571,A 0.000,B 0.000,C 90.000,E1 282.827} C_DIS
LIN {X -0.030,Y -461.311,Z 947.564,A 0.000,B 0.000,C 90.000,E1 281.535} C_DIS
LIN {X 0.135,Y -468.820,Z 947.558,A 0.000,B 0.000,C 90.000,E1 280.489} C_DIS
LIN {X -0.071,Y -475.573,Z 947.553,A 0.000,B 0.000,C 90.000,E1 279.500} C_DIS
LIN {X -0.076,Y -479.967,Z 947.549,A 0.000,B 0.000,C 90.000,E1 278.746} C_DIS
LIN {X -0.045,Y -483.663,Z 947.544,A 0.000,B 0.000,C 90.000,E1 277.992} C_DIS
LIN {X 0.133,Y -485.714,Z 947.542,A 0.000,B 0.000,C 90.000,E1 277.473} C_DIS
LIN {X -0.097,Y -487.458,Z 947.539,A 0.000,B 0.000,C 90.000,E1 277.004} C_DIS
LIN {X 0.100,Y -488.883,Z 947.536,A 0.000,B 0.000,C 90.000,E1 276.486} C_DIS
LIN {X -0.181,Y -490.005,Z 947.533,A 0.000,B 0.000,C 90.000,E1 276.024} C_DIS
LIN {X -0.014,Y -490.798,Z 947.531,A 0.000,B 0.000,C 90.000,E1 275.511} C_DIS
LIN {X 0.211,Y -491.190,Z 947.528,A 0.000,B 0.000,C 90.000,E1 274.992} C_DIS
LIN {X -0.052,Y -491.222,Z 947.525,A 0.000,B 0.000,C 90.000,E1 274.531} C_DIS
LIN {X 0.175,Y -490.806,Z 947.522,A 0.000,B 0.000,C 90.000,E1 274.012} C_DIS
LIN {X -0.122,Y -489.814,Z 947.520,A 0.000,B 0.000,C 90.000,E1 273.555} C_DIS
LIN {X 0.099,Y -488.301,Z 947.517,A 0.000,B 0.000,C 90.000,E1 273.037} C_DIS
LIN {X -0.200,Y -486.163,Z 947.514,A 0.000,B 0.000,C 90.000,E1 272.579} C_DIS
LIN {X -0.018,Y -483.292,Z 947.511,A 0.000,B 0.000,C 90.000,E1 272.064} C_DIS
LIN {X -0.177,Y -481.600,Z 947.510,A 0.000,B 0.000,C 90.000,E1 271.835} C_DIS
LIN {X -0.010,Y -477.450,Z 947.507,A 0.000,B 0.000,C 90.000,E1 271.318} C_DIS
LIN {X 0.140,Y -472.323,Z 947.505,A 0.000,B 0.000,C 90.000,E1 270.802} C_DIS
LIN {X 0.057,Y -466.528,Z 947.502,A 0.000,B 0.000,C 90.000,E1 270.344} C_DIS
LIN {X -0.082,Y -460.376,Z 947.500,A 0.000,B 0.000,C 90.000,E1 269.943} C_DIS
LIN {X 0.181,Y -453.891,Z 947.498,A 0.000,B 0.000,C 90.000,E1 269.542} C_DIS
LIN {X -0.046,Y -447.055,Z 947.496,A 0.000,B 0.000,C 90.000,E1 269.255} C_DIS
LIN {X 0.112,Y -440.042,Z 947.494,A 0.000,B 0.000,C 90.000,E1 268.969} C_DIS
LIN {X 0.171,Y -432.819,Z 947.493,A 0.000,B 0.000,C 90.000,E1 268.740} C_DIS
LIN {X 0.096,Y -425.420,Z 947.492,A 0.000,B 0.000,C 90.000,E1 268.568} C_DIS
LIN {X -0.119,Y -417.194,Z 947.491,A 0.000,B 0.000,C 90.000,E1 268.453} C_DIS
LIN {X 0.100,Y -408.443,Z 947.491,A 0.000,B 0.000,C 90.000,E1 268.339} C_DIS
LIN {X -0.057,Y -402.184,Z 947.491,A 0.000,B 0.000,C 90.000,E1 268.339} C_DIS
LIN {X -0.060,Y -181.180,Z 947.491,A 0.000,B 0.000,C 90.000,E1 268.339} C_DIS
LIN {X 0.072,Y -180.841,Z 947.472,A 0.000,B 0.000,C 90.000,E1 264.894} C_DIS
LIN {X -0.025,Y -178.949,Z 947.444,A 0.000,B 0.000,C 90.000,E1 259.859} C_DIS
LIN {X -0.008,Y -176.852,Z 947.425,A 0.000,B 0.000,C 90.000,E1 256.464} C_DIS
LIN {X -0.037,Y -175.511,Z 947.411,A 0.000,B 0.000,C 90.000,E1 253.921} C_DIS
LIN {X 0.026,Y -172.251,Z 947.387,A 0.000,B 0.000,C 90.000,E1 249.625} C_DIS
LIN {X 0.005,Y -171.729,Z 947.382,A 0.000,B 0.000,C 90.000,E1 248.773} C_DIS
LIN {X 0.013,Y -167.325,Z 947.353,A 0.000,B 0.000,C 90.000,E1 243.589} C_DIS
LIN {X -0.055,Y -166.709,Z 947.348,A 0.000,B 0.000,C 90.000,E1 242.743} C_DIS
LIN {X 0.083,Y -162.689,Z 947.324,A 0.000,B 0.000,C 90.000,E1 238.329} C_DIS
LIN {X -0.079,Y -161.380,Z 947.314,A 0.000,B 0.000,C 90.000,E1 236.628} C_DIS
LIN {X -0.036,Y -157.373,Z 947.290,A 0.000,B 0.000,C 90.000,E1 232.190} C_DIS
LIN {X -0.001,Y -155.366,Z 947.275,A 0.000,B 0.000,C 90.000,E1 229.504} C_DIS
LIN {X 0.046,Y -151.706,Z 947.250,A 0.000,B 0.000,C 90.000,E1 225.000} C_DIS
LIN {X 0.056,Y -149.897,Z 947.235,A 0.000,B 0.000,C 90.000,E1 222.285} C_DIS
LIN {X 0.080,Y -146.757,Z 947.210,A 0.000,B 0.000,C 90.000,E1 217.729} C_DIS
LIN {X -0.022,Y -145.324,Z 947.195,A 0.000,B 0.000,C 90.000,E1 215.025} C_DIS
LIN {X 0.017,Y -142.408,Z 947.164,A 0.000,B 0.000,C 90.000,E1 209.489} C_DIS
LIN {X -0.056,Y -141.392,Z 947.148,A 0.000,B 0.000,C 90.000,E1 206.744} C_DIS
LIN {X -0.069,Y -139.352,Z 947.112,A 0.000,B 0.000,C 90.000,E1 200.248} C_DIS
LIN {X 0.052,Y -138.791,Z 947.097,A 0.000,B 0.000,C 90.000,E1 197.402} C_DIS
LIN {X -0.025,Y -138.346,Z 947.055,A 0.000,B 0.000,C 90.000,E1 189.962} C_DIS
LIN {X -0.008,Y -139.380,Z 947.009,A 0.000,B 0.000,C 90.000,E1 181.547} C_DIS
LIN {X 0.045,Y -141.273,Z 946.972,A 0.000,B 0.000,C 90.000,E1 175.008} C_DIS
LIN {X 0.003,Y -142.638,Z 946.957,A 0.000,B 0.000,C 90.000,E1 172.243} C_DIS
LIN {X -0.046,Y -144.968,Z 946.931,A 0.000,B 0.000,C 90.000,E1 167.645} C_DIS
LIN {X -0.055,Y -147.596,Z 946.911,A 0.000,B 0.000,C 90.000,E1 163.976} C_DIS
LIN {X -0.026,Y -150.214,Z 946.891,A 0.000,B 0.000,C 90.000,E1 160.315} C_DIS
LIN {X 0.041,Y -153.600,Z 946.870,A 0.000,B 0.000,C 90.000,E1 156.666} C_DIS
LIN {X 0.030,Y -157.017,Z 946.850,A 0.000,B 0.000,C 90.000,E1 153.076} C_DIS
LIN {X -0.039,Y -161.137,Z 946.831,A 0.000,B 0.000,C 90.000,E1 149.537} C_DIS
LIN {X 0.044,Y -163.236,Z 946.821,A 0.000,B 0.000,C 90.000,E1 147.740} C_DIS
LIN {X -0.090,Y -167.670,Z 946.801,A 0.000,B 0.000,C 90.000,E1 144.276} C_DIS
LIN {X 0.058,Y -171.493,Z 946.787,A 0.000,B 0.000,C 90.000,E1 141.618} C_DIS
LIN {X 0.103,Y -176.425,Z 946.768,A 0.000,B 0.000,C 90.000,E1 138.162} C_DIS
LIN {X -0.026,Y -180.720,Z 946.754,A 0.000,B 0.000,C 90.000,E1 135.648} C_DIS
LIN {X -0.045,Y -186.124,Z 946.735,A 0.000,B 0.000,C 90.000,E1 132.285} C_DIS
LIN {X 0.012,Y -190.762,Z 946.721,A 0.000,B 0.000,C 90.000,E1 129.769} C_DIS
LIN {X -0.032,Y -194.462,Z 946.709,A 0.000,B 0.000,C 90.000,E1 127.604} C_DIS
LIN {X -0.101,Y -297.445,Z 946.709,A 0.000,B 0.000,C 90.000,E1 127.604} C_DIS
LIN {X -0.006,Y -301.878,Z 946.708,A 0.000,B 0.000,C 90.000,E1 127.443} C_DIS
LIN {X -0.094,Y -304.049,Z 946.707,A 0.000,B 0.000,C 90.000,E1 127.317} C_DIS
LIN {X 0.177,Y -307.921,Z 946.705,A 0.000,B 0.000,C 90.000,E1 126.870} C_DIS
LIN {X 0.169,Y -311.392,Z 946.702,A 0.000,B 0.000,C 90.000,E1 126.297} C_DIS
LIN {X -0.047,Y -312.776,Z 946.700,A 0.000,B 0.000,C 90.000,E1 126.011} C_DIS
LIN {X -0.018,Y -324.325,Z 946.680,A 0.000,B 0.000,C 90.000,E1 122.467} C_DIS
LIN {X 0.051,Y -335.083,Z 946.665,A 0.000,B 0.000,C 90.000,E1 119.617} C_DIS
LIN {X -0.195,Y -347.220,Z 946.649,A 0.000,B 0.000,C 90.000,E1 116.873} C_DIS
LIN {X -0.111,Y -360.835,Z 946.634,A 0.000,B 0.000,C 90.000,E1 114.131} C_DIS
LIN {X 0.163,Y -374.282,Z 946.621,A 0.000,B 0.000,C 90.000,E1 111.716} C_DIS
LIN {X 0.170,Y -389.091,Z 946.608,A 0.000,B 0.000,C 90.000,E1 109.396} C_DIS
LIN {X 0.037,Y -405.368,Z 946.595,A 0.000,B 0.000,C 90.000,E1 107.149} C_DIS
LIN {X -0.064,Y -423.230,Z 946.583,A 0.000,B 0.000,C 90.000,E1 104.954} C_DIS
LIN {X -0.158,Y -442.692,Z 946.571,A 0.000,B 0.000,C 90.000,E1 102.827} C_DIS
LIN {X -0.103,Y -462.947,Z 946.560,A 0.000,B 0.000,C 90.000,E1 100.838} C_DIS
LIN {X -0.087,Y -467.968,Z 946.558,A 0.000,B 0.000,C 90.000,E1 100.366} C_DIS
LIN {X -0.142,Y -469.841,Z 946.556,A 0.000,B 0.000,C 90.000,E1 100.141} C_DIS
LIN {X 0.173,Y -471.392,Z 946.555,A 0.000,B 0.000,C 90.000,E1 99.849} C_DIS
LIN {X 0.022,Y -472.554,Z 946.553,A 0.000,B 0.000,C 90.000,E1 99.613} C_DIS
LIN {X 0.129,Y -473.957,Z 946.551,A 0.000,B 0.000,C 90.000,E1 99.095} C_DIS
LIN {X -0.152,Y -474.332,Z 946.548,A 0.000,B 0.000,C 90.000,E1 98.624} C_DIS
LIN {X -0.030,Y -473.746,Z 946.545,A 0.000,B 0.000,C 90.000,E1 98.106} C_DIS
LIN {X 0.097,Y -472.108,Z 946.542,A 0.000,B 0.000,C 90.000,E1 97.587} C_DIS
LIN {X -0.044,Y -470.805,Z 946.541,A 0.000,B 0.000,C 90.000,E1 97.352} C_DIS
LIN {X 0.070,Y -455.918,Z 946.528,A 0.000,B 0.000,C 90.000,E1 95.049} C_DIS
LIN {X 0.058,Y -446.155,Z 946.519,A 0.000,B 0.000,C 90.000,E1 93.498} C_DIS
LIN {X -0.084,Y -431.349,Z 946.506,A 0.000,B 0.000,C 90.000,E1 91.146} C_DIS
LIN {X 0.024,Y -414.124,Z 946.490,A 0.000,B 0.000,C 90.000,E1 88.165} C_DIS
LIN {X 0.117,Y -404.905,Z 946.481,A 0.000,B 0.000,C 90.000,E1 86.502} C_DIS
LIN {X 0.150,Y -392.526,Z 946.468,A 0.000,B 0.000,C 90.000,E1 84.261} C_DIS
LIN {X -0.088,Y -383.180,Z 946.459,A 0.000,B 0.000,C 90.000,E1 82.591} C_DIS
LIN {X -0.009,Y -373.559,Z 946.449,A 0.000,B 0.000,C 90.000,E1 80.849} C_DIS
LIN {X -0.099,Y -363.778,Z 946.439,A 0.000,B 0.000,C 90.000,E1 79.106} C_DIS
LIN {X 0.048,Y -353.672,Z 946.429,A 0.000,B 0.000,C 90.000,E1 77.297} C_DIS
LIN {X -0.019,Y -338.619,Z 946.414,A 0.000,B 0.000,C 90.000,E1 74.574} C_DIS
LIN {X -0.065,Y -321.610,Z 946.395,A 0.000,B 0.000,C 90.000,E1 71.148} C_DIS
LIN {X -0.013,Y -311.140,Z 946.383,A 0.000,B 0.000,C 90.000,E1 68.901} C_DIS
LIN {X 0.031,Y -300.673,Z 946.370,A 0.000,B 0.000,C 90.000,E1 66.613} C_DIS
LIN {X 0.068,Y -288.747,Z 946.355,A 0.000,B 0.000,C 90.000,E1 63.948} C_DIS
LIN {X -0.019,Y -278.366,Z 946.342,A 0.000,B 0.000,C 90.000,E1 61.591} C_DIS
LIN {X -0.016,Y -266.613,Z 946.327,A 0.000,B 0.000,C 90.000,E1 58.820} C_DIS
LIN {X 0.142,Y -253.947,Z 946.309,A 0.000,B 0.000,C 90.000,E1 55.595} C_DIS
LIN {X 0.025,Y -242.286,Z 946.291,A 0.000,B 0.000,C 90.000,E1 52.351} C_DIS
LIN {X -0.003,Y -231.563,Z 946.272,A 0.000,B 0.000,C 90.000,E1 49.013} C_DIS
LIN {X 0.024,Y -222.675,Z 946.255,A 0.000,B 0.000,C 90.000,E1 45.972} C_DIS
LIN {X 0.006,Y -214.404,Z 946.238,A 0.000,B 0.000,C 90.000,E1 42.894} C_DIS
LIN {X -0.038,Y -206.765,Z 946.221,A 0.000,B 0.000,C 90.000,E1 39.769} C_DIS
LIN {X -0.049,Y -199.672,Z 946.203,A 0.000,B 0.000,C 90.000,E1 36.583} C_DIS
LIN {X 0.129,Y -193.172,Z 946.185,A 0.000,B 0.000,C 90.000,E1 33.293} C_DIS
LIN {X -0.013,Y -187.322,Z 946.167,A 0.000,B 0.000,C 90.000,E1 30.050} C_DIS
LIN {X -0.082,Y -182.107,Z 946.148,A 0.000,B 0.000,C 90.000,E1 26.744} C_DIS
LIN {X 0.054,Y -177.581,Z 946.130,A 0.000,B 0.000,C 90.000,E1 23.334} C_DIS
LIN {X 0.033,Y -173.721,Z 946.111,A 0.000,B 0.000,C 90.000,E1 19.939} C_DIS
LIN {X -0.018,Y -169.857,Z 946.087,A 0.000,B 0.000,C 90.000,E1 15.662} C_DIS
LIN {X 0.078,Y -167.133,Z 946.063,A 0.000,B 0.000,C 90.000,E1 11.299} C_DIS
LIN {X 0.003,Y -165.036,Z 946.029,A 0.000,B 0.000,C 90.000,E1 5.220} C_DIS
LIN {X 0.065,Y -166.292,Z 945.968,A 0.000,B 0.000,C 90.000,E1 354.261} C_DIS
LIN {X 0.025,Y -169.191,Z 945.939,A 0.000,B 0.000,C 90.000,E1 349.050} C_DIS
LIN {X 0.020,Y -172.005,Z 945.920,A 0.000,B 0.000,C 90.000,E1 345.589} C_DIS
LIN {X 0.080,Y -176.519,Z 945.896,A 0.000,B 0.000,C 90.000,E1 341.275} C_DIS
LIN {X -0.072,Y -180.889,Z 945.877,A 0.000,B 0.000,C 90.000,E1 337.922} C_DIS
LIN {X -0.014,Y -185.968,Z 945.859,A 0.000,B 0.000,C 90.000,E1 334.537} C_DIS
LIN {X 0.084,Y -191.764,Z 945.840,A 0.000,B 0.000,C 90.000,E1 331.179} C_DIS
LIN {X 0.017,Y -198.204,Z 945.822,A 0.000,B 0.000,C 90.000,E1 327.916} C_DIS
LIN {X -0.017,Y -205.236,Z 945.804,A 0.000,B 0.000,C 90.000,E1 324.689} C_DIS
LIN {X 0.019,Y -212.827,Z 945.786,A 0.000,B 0.000,C 90.000,E1 321.492} C_DIS
LIN {X -0.001,Y -220.988,Z 945.769,A 0.000,B 0.000,C 90.000,E1 318.366} C_DIS
LIN {X -0.124,Y -230.052,Z 945.752,A 0.000,B 0.000,C 90.000,E1 315.324} C_DIS
LIN {X -0.026,Y -240.208,Z 945.735,A 0.000,B 0.000,C 90.000,E1 312.285} C_DIS
LIN {X -0.134,Y -250.131,Z 945.721,A 0.000,B 0.000,C 90.000,E1 309.725} C_DIS
LIN {X -0.053,Y -258.013,Z 945.710,A 0.000,B 0.000,C 90.000,E1 307.890} C_DIS
LIN {X -0.026,Y -270.315,Z 945.697,A 0.000,B 0.000,C 90.000,E1 305.391} C_DIS
LIN {X 0.032,Y -287.908,Z 945.679,A 0.000,B 0.000,C 90.000,E1 302.260} C_DIS
LIN {X -0.166,Y -306.942,Z 945.663,A 0.000,B 0.000,C 90.000,E1 299.283} C_DIS
LIN {X -0.049,Y -320.664,Z 945.652,A 0.000,B 0.000,C 90.000,E1 297.308} C_DIS
LIN {X 0.005,Y -338.639,Z 945.639,A 0.000,B 0.000,C 90.000,E1 295.079} C_DIS
LIN {X -0.059,Y -357.370,Z 945.628,A 0.000,B 0.000,C 90.000,E1 293.003} C_DIS
LIN {X -0.096,Y -378.798,Z 945.615,A 0.000,B 0.000,C 90.000,E1 290.791} C_DIS
LIN {X -0.056,Y -392.129,Z 945.608,A 0.000,B 0.000,C 90.000,E1 289.450} C_DIS
LIN {X -0.125,Y -405.073,Z 945.601,A 0.000,B 0.000,C 90.000,E1 288.127} C_DIS
LIN {X 0.098,Y -415.147,Z 945.595,A 0.000,B 0.000,C 90.000,E1 287.040} C_DIS
LIN {X -0.004,Y -425.050,Z 945.589,A 0.000,B 0.000,C 90.000,E1 285.969} C_DIS
LIN {X -0.072,Y -434.410,Z 945.583,A 0.000,B 0.000,C 90.000,E1 284.898} C_DIS
LIN {X -0.033,Y -443.166,Z 945.577,A 0.000,B 0.000,C 90.000,E1 283.828} C_DIS
LIN {X -0.193,Y -453.633,Z 945.570,A 0.000,B 0.000,C 90.000,E1 282.535} C_DIS
LIN {X -0.033,Y -461.620,Z 945.564,A 0.000,B 0.000,C 90.000,E1 281.478} C_DIS
LIN {X 0.137,Y -469.096,Z 945.558,A 0.000,B 0.000,C 90.000,E1 280.433} C_DIS
LIN {X -0.064,Y -475.823,Z 945.552,A 0.000,B 0.000,C 90.000,E1 279.443} C_DIS
LIN {X 0.136,Y -478.844,Z 945.550,A 0.000,B 0.000,C 90.000,E1 278.916} C_DIS
LIN {X 0.159,Y -482.701,Z 945.545,A 0.000,B 0.000,C 90.000,E1 278.163} C_DIS
LIN {X 0.212,Y -485.880,Z 945.541,A 0.000,B 0.000,C 90.000,E1 277.409} C_DIS
LIN {X -0.086,Y -487.622,Z 945.539,A 0.000,B 0.000,C 90.000,E1 276.947} C_DIS
LIN {X 0.112,Y -489.025,Z 945.536,A 0.000,B 0.000,C 90.000,E1 276.429} C_DIS
LIN {X -0.167,Y -490.142,Z 945.533,A 0.000,B 0.000,C 90.000,E1 275.967} C_DIS
LIN {X 0.001,Y -490.888,Z 945.530,A 0.000,B 0.000,C 90.000,E1 275.454} C_DIS
LIN {X 0.228,Y -491.253,Z 945.528,A 0.000,B 0.000,C 90.000,E1 274.935} C_DIS
LIN {X -0.035,Y -491.249,Z 945.525,A 0.000,B 0.000,C 90.000,E1 274.473} C_DIS
LIN {X 0.192,Y -490.793,Z 945.522,A 0.000,B 0.000,C 90.000,E1 273.955} C_DIS
LIN {X -0.104,Y -489.756,Z 945.519,A 0.000,B 0.000,C 90.000,E1 273.498} C_DIS
LIN {X 0.116,Y -488.193,Z 945.517,A 0.000,B 0.000,C 90.000,E1 272.980} C_DIS
LIN {X -0.182,Y -485.986,Z 945.514,A 0.000,B 0.000,C 90.000,E1 272.522} C_DIS
LIN {X -0.006,Y -483.062,Z 945.511,A 0.000,B 0.000,C 90.000,E1 272.007} C_DIS
LIN {X 0.169,Y -479.360,Z 945.508,A 0.000,B 0.000,C 90.000,E1 271.489} C_DIS
LIN {X -0.168,Y -474.612,Z 945.506,A 0.000,B 0.000,C 90.000,E1 271.031} C_DIS
LIN {X 0.027,Y -468.971,Z 945.503,A 0.000,B 0.000,C 90.000,E1 270.516} C_DIS
LIN {X 0.195,Y -462.976,Z 945.500,A 0.000,B 0.000,C 90.000,E1 270.057} C_DIS
LIN {X -0.166,Y -456.569,Z 945.498,A 0.000,B 0.000,C 90.000,E1 269.714} C_DIS
LIN {X -0.097,Y -449.865,Z 945.496,A 0.000,B 0.000,C 90.000,E1 269.370} C_DIS
LIN {X -0.068,Y -443.045,Z 945.495,A 0.000,B 0.000,C 90.000,E1 269.083} C_DIS
LIN {X -0.158,Y -435.931,Z 945.494,A 0.000,B 0.000,C 90.000,E1 268.854} C_DIS
LIN {X 0.079,Y -428.601,Z 945.492,A 0.000,B 0.000,C 90.000,E1 268.625} C_DIS
LIN {X 0.161,Y -420.999,Z 945.492,A 0.000,B 0.000,C 90.000,E1 268.453} C_DIS
LIN {X 0.087,Y -411.578,Z 945.491,A 0.000,B 0.000,C 90.000,E1 268.339} C_DIS
LIN {X -0.135,Y -405.780,Z 945.491,A 0.000,B 0.000,C 90.000,E1 268.339} C_DIS
LIN {X 0.088,Y -181.178,Z 945.491,A 0.000,B 0.000,C 90.000,E1 268.282} C_DIS
LIN {X 0.011,Y -180.836,Z 945.472,A 0.000,B 0.000,C 90.000,E1 264.894} C_DIS
LIN {X 0.091,Y -178.942,Z 945.443,A 0.000,B 0.000,C 90.000,E1 259.803} C_DIS
LIN {X -0.042,Y -175.993,Z 945.415,A 0.000,B 0.000,C 90.000,E1 254.755} C_DIS
LIN {X -0.096,Y -175.496,Z 945.411,A 0.000,B 0.000,C 90.000,E1 253.921} C_DIS
LIN {X -0.033,Y -172.239,Z 945.387,A 0.000,B 0.000,C 90.000,E1 249.625} C_DIS
LIN {X -0.054,Y -171.716,Z 945.382,A 0.000,B 0.000,C 90.000,E1 248.773} C_DIS
LIN {X -0.044,Y -167.311,Z 945.353,A 0.000,B 0.000,C 90.000,E1 243.589} C_DIS
LIN {X 0.036,Y -166.693,Z 945.348,A 0.000,B 0.000,C 90.000,E1 242.692} C_DIS
LIN {X 0.026,Y -162.674,Z 945.324,A 0.000,B 0.000,C 90.000,E1 238.329} C_DIS
LIN {X 0.000,Y -161.364,Z 945.314,A 0.000,B 0.000,C 90.000,E1 236.580} C_DIS
LIN {X -0.091,Y -157.357,Z 945.290,A 0.000,B 0.000,C 90.000,E1 232.190} C_DIS
LIN {X 0.062,Y -155.346,Z 945.275,A 0.000,B 0.000,C 90.000,E1 229.461} C_DIS
LIN {X -0.008,Y -151.693,Z 945.250,A 0.000,B 0.000,C 90.000,E1 225.000} C_DIS
LIN {X 0.039,Y -150.554,Z 945.240,A 0.000,B 0.000,C 90.000,E1 223.176} C_DIS
LIN {X -0.043,Y -147.281,Z 945.215,A 0.000,B 0.000,C 90.000,E1 218.669} C_DIS
LIN {X -0.076,Y -145.310,Z 945.194,A 0.000,B 0.000,C 90.000,E1 215.025} C_DIS
LIN {X 0.036,Y -142.400,Z 945.164,A 0.000,B 0.000,C 90.000,E1 209.461} C_DIS
LIN {X 0.018,Y -141.382,Z 945.148,A 0.000,B 0.000,C 90.000,E1 206.693} C_DIS
LIN {X 0.059,Y -139.349,Z 945.112,A 0.000,B 0.000,C 90.000,E1 200.174} C_DIS
LIN {X 0.001,Y -138.786,Z 945.097,A 0.000,B 0.000,C 90.000,E1 197.402} C_DIS
LIN {X 0.059,Y -138.344,Z 945.055,A 0.000,B 0.000,C 90.000,E1 189.905} C_DIS
LIN {X -0.060,Y -139.386,Z 945.008,A 0.000,B 0.000,C 90.000,E1 181.547} C_DIS
LIN {X -0.007,Y -141.283,Z 944.972,A 0.000,B 0.000,C 90.000,E1 175.008} C_DIS
LIN {X -0.049,Y -142.646,Z 944.957,A 0.000,B 0.000,C 90.000,E1 172.243} C_DIS
LIN {X 0.043,Y -144.982,Z 944.931,A 0.000,B 0.000,C 90.000,E1 167.589} C_DIS
LIN {X 0.034,Y -147.609,Z 944.911,A 0.000,B 0.000,C 90.000,E1 163.921} C_DIS
LIN {X -0.029,Y -150.231,Z 944.890,A 0.000,B 0.000,C 90.000,E1 160.296} C_DIS
LIN {X -0.014,Y -153.622,Z 944.870,A 0.000,B 0.000,C 90.000,E1 156.666} C_DIS
LIN {X -0.026,Y -157.038,Z 944.850,A 0.000,B 0.000,C 90.000,E1 153.076} C_DIS
LIN {X -0.095,Y -161.163,Z 944.831,A 0.000,B 0.000,C 90.000,E1 149.537} C_DIS
LIN {X -0.013,Y -163.259,Z 944.821,A 0.000,B 0.000,C 90.000,E1 147.740} C_DIS
LIN {X 0.086,Y -167.698,Z 944.801,A 0.000,B 0.000,C 90.000,E1 144.196} C_DIS
LIN {X -0.001,Y -171.519,Z 944.787,A 0.000,B 0.000,C 90.000,E1 141.618} C_DIS
LIN {X 0.042,Y -176.456,Z 944.768,A 0.000,B 0.000,C 90.000,E1 138.162} C_DIS
LIN {X -0.087,Y -180.752,Z 944.753,A 0.000,B 0.000,C 90.000,E1 135.648} C_DIS
LIN {X 0.031,Y -186.158,Z 944.735,A 0.000,B 0.000,C 90.000,E1 132.243} C_DIS
LIN {X 0.096,Y -190.795,Z 944.721,A 0.000,B 0.000,C 90.000,E1 129.725} C_DIS
LIN {X 0.072,Y -194.407,Z 944.709,A 0.000,B 0.000,C 90.000,E1 127.604} C_DIS
LIN {X 0.081,Y -296.467,Z 944.709,A 0.000,B 0.000,C 90.000,E1 127.604} C_DIS
LIN {X 0.020,Y -297.792,Z 944.709,A 0.000,B 0.000,C 90.000,E1 127.604} C_DIS
LIN {X 0.007,Y -302.253,Z 944.708,A 0.000,B 0.000,C 90.000,E1 127.443} C_DIS
LIN {X -0.008,Y -304.537,Z 944.707,A 0.000,B 0.000,C 90.000,E1 127.282} C_DIS
LIN {X -0.093,Y -308.403,Z 944.705,A 0.000,B 0.000,C 90.000,E1 126.870} C_DIS
LIN {X 0.056,Y -310.309,Z 944.703,A 0.000,B 0.000,C 90.000,E1 126.537} C_DIS
LIN {X 0.143,Y -311.808,Z 944.701,A 0.000,B 0.000,C 90.000,E1 126.217} C_DIS
LIN {X -0.066,Y -313.075,Z 944.700,A 0.000,B 0.000,C 90.000,E1 125.931} C_DIS
LIN {X -0.201,Y -324.589,Z 944.680,A 0.000,B 0.000,C 90.000,E1 122.418} C_DIS
LIN {X 0.044,Y -335.385,Z 944.664,A 0.000,B 0.000,C 90.000,E1 119.539} C_DIS
LIN {X 0.109,Y -347.561,Z 944.649,A 0.000,B 0.000,C 90.000,E1 116.744} C_DIS
LIN {X 0.068,Y -361.221,Z 944.634,A 0.000,B 0.000,C 90.000,E1 114.027} C_DIS
LIN {X 0.022,Y -374.709,Z 944.620,A 0.000,B 0.000,C 90.000,E1 111.663} C_DIS
LIN {X 0.169,Y -389.563,Z 944.607,A 0.000,B 0.000,C 90.000,E1 109.322} C_DIS
LIN {X -0.082,Y -405.888,Z 944.595,A 0.000,B 0.000,C 90.000,E1 107.094} C_DIS
LIN {X -0.170,Y -423.803,Z 944.583,A 0.000,B 0.000,C 90.000,E1 104.898} C_DIS
LIN {X -0.241,Y -443.307,Z 944.571,A 0.000,B 0.000,C 90.000,E1 102.771} C_DIS
LIN {X -0.143,Y -463.580,Z 944.560,A 0.000,B 0.000,C 90.000,E1 100.782} C_DIS
LIN {X -0.116,Y -468.477,Z 944.557,A 0.000,B 0.000,C 90.000,E1 100.310} C_DIS
LIN {X -0.082,Y -470.224,Z 944.556,A 0.000,B 0.000,C 90.000,E1 100.074} C_DIS
LIN {X 0.152,Y -471.679,Z 944.555,A 0.000,B 0.000,C 90.000,E1 99.792} C_DIS
LIN {X 0.003,Y -472.763,Z 944.553,A 0.000,B 0.000,C 90.000,E1 99.557} C_DIS
LIN {X 0.186,Y -474.042,Z 944.550,A 0.000,B 0.000,C 90.000,E1 99.029} C_DIS
LIN {X -0.169,Y -474.311,Z 944.547,A 0.000,B 0.000,C 90.000,E1 98.568} C_DIS
LIN {X -0.044,Y -473.614,Z 944.545,A 0.000,B 0.000,C 90.000,E1 98.049} C_DIS
LIN {X 0.084,Y -471.844,Z 944.542,A 0.000,B 0.000,C 90.000,E1 97.530} C_DIS
LIN {X -0.059,Y -470.455,Z 944.540,A 0.000,B 0.000,C 90.000,E1 97.296} C_DIS
LIN {X 0.050,Y -455.591,Z 944.528,A 0.000,B 0.000,C 90.000,E1 94.992} C_DIS
LIN {X 0.034,Y -445.859,Z 944.519,A 0.000,B 0.000,C 90.000,E1 93.440} C_DIS
LIN {X 0.167,Y -432.711,Z 944.507,A 0.000,B 0.000,C 90.000,E1 91.318} C_DIS
LIN {X -0.124,Y -415.364,Z 944.491,A 0.000,B 0.000,C 90.000,E1 88.396} C_DIS
LIN {X 0.007,Y -406.164,Z 944.482,A 0.000,B 0.000,C 90.000,E1 86.731} C_DIS
LIN {X 0.016,Y -395.313,Z 944.471,A 0.000,B 0.000,C 90.000,E1 84.780} C_DIS
LIN {X -0.133,Y -384.414,Z 944.460,A 0.000,B 0.000,C 90.000,E1 82.818} C_DIS
LIN {X -0.082,Y -374.817,Z 944.450,A 0.000,B 0.000,C 90.000,E1 81.084} C_DIS
LIN {X -0.151,Y -365.069,Z 944.441,A 0.000,B 0.000,C 90.000,E1 79.342} C_DIS
LIN {X 0.066,Y -356.726,Z 944.432,A 0.000,B 0.000,C 90.000,E1 77.825} C_DIS
LIN {X 0.079,Y -343.228,Z 944.419,A 0.000,B 0.000,C 90.000,E1 75.408} C_DIS
LIN {X 0.108,Y -327.299,Z 944.402,A 0.000,B 0.000,C 90.000,E1 72.308} C_DIS
LIN {X -0.025,Y -316.805,Z 944.390,A 0.000,B 0.000,C 90.000,E1 70.115} C_DIS
LIN {X 0.035,Y -306.320,Z 944.377,A 0.000,B 0.000,C 90.000,E1 67.847} C_DIS
LIN {X 0.089,Y -297.371,Z 944.366,A 0.000,B 0.000,C 90.000,E1 65.869} C_DIS
LIN {X -0.072,Y -286.978,Z 944.353,A 0.000,B 0.000,C 90.000,E1 63.563} C_DIS
LIN {X -0.055,Y -276.586,Z 944.340,A 0.000,B 0.000,C 90.000,E1 61.179} C_DIS
LIN {X -0.034,Y -263.401,Z 944.322,A 0.000,B 0.000,C 90.000,E1 58.043} C_DIS
LIN {X 0.046,Y -250.939,Z 944.305,A 0.000,B 0.000,C 90.000,E1 54.815} C_DIS
LIN {X 0.001,Y -239.551,Z 944.286,A 0.000,B 0.000,C 90.000,E1 51.537} C_DIS
LIN {X 0.052,Y -229.023,Z 944.268,A 0.000,B 0.000,C 90.000,E1 48.162} C_DIS
LIN {X 0.027,Y -220.324,Z 944.251,A 0.000,B 0.000,C 90.000,E1 45.121} C_DIS
LIN {X -0.045,Y -212.269,Z 944.234,A 0.000,B 0.000,C 90.000,E1 42.043} C_DIS
LIN {X -0.112,Y -204.846,Z 944.216,A 0.000,B 0.000,C 90.000,E1 38.910} C_DIS
LIN {X -0.002,Y -197.945,Z 944.198,A 0.000,B 0.000,C 90.000,E1 35.678} C_DIS
LIN {X 0.027,Y -191.633,Z 944.180,A 0.000,B 0.000,C 90.000,E1 32.418} C_DIS
LIN {X 0.012,Y -185.973,Z 944.162,A 0.000,B 0.000,C 90.000,E1 29.127} C_DIS
LIN {X -0.011,Y -180.931,Z 944.143,A 0.000,B 0.000,C 90.000,E1 25.796} C_DIS
LIN {X 0.026,Y -176.634,Z 944.125,A 0.000,B 0.000,C 90.000,E1 22.408} C_DIS
LIN {X -0.091,Y -172.130,Z 944.101,A 0.000,B 0.000,C 90.000,E1 18.181} C_DIS
LIN {X 0.042,Y -168.774,Z 944.077,A 0.000,B 0.000,C 90.000,E1 13.828} C_DIS
LIN {X 0.017,Y -166.160,Z 944.048,A 0.000,B 0.000,C 90.000,E1 8.624} C_DIS
LIN {X -0.035,Y -165.897,Z 943.978,A 0.000,B 0.000,C 90.000,E1 356.045} C_DIS
LIN {X 0.026,Y -168.295,Z 943.949,A 0.000,B 0.000,C 90.000,E1 350.792} C_DIS
LIN {X 0.006,Y -171.468,Z 943.925,A 0.000,B 0.000,C 90.000,E1 346.464} C_DIS
LIN {X -0.045,Y -175.789,Z 943.901,A 0.000,B 0.000,C 90.000,E1 342.181} C_DIS
LIN {X -0.047,Y -179.988,Z 943.882,A 0.000,B 0.000,C 90.000,E1 338.773} C_DIS
LIN {X 0.088,Y -184.894,Z 943.863,A 0.000,B 0.000,C 90.000,E1 335.357} C_DIS
LIN {X 0.076,Y -190.485,Z 943.845,A 0.000,B 0.000,C 90.000,E1 332.025} C_DIS
LIN {X 0.045,Y -196.771,Z 943.826,A 0.000,B 0.000,C 90.000,E1 328.742} C_DIS
LIN {X -0.026,Y -203.644,Z 943.808,A 0.000,B 0.000,C 90.000,E1 325.515} C_DIS
LIN {X -0.022,Y -211.157,Z 943.791,A 0.000,B 0.000,C 90.000,E1 322.316} C_DIS
LIN {X -0.036,Y -219.106,Z 943.773,A 0.000,B 0.000,C 90.000,E1 319.175} C_DIS
LIN {X 0.107,Y -227.935,Z 943.756,A 0.000,B 0.000,C 90.000,E1 316.053} C_DIS
LIN {X -0.014,Y -237.799,Z 943.739,A 0.000,B 0.000,C 90.000,E1 313.056} C_DIS
LIN {X -0.021,Y -248.866,Z 943.723,A 0.000,B 0.000,C 90.000,E1 310.092} C_DIS
LIN {X 0.048,Y -256.559,Z 943.713,A 0.000,B 0.000,C 90.000,E1 308.257} C_DIS
LIN {X 0.041,Y -268.606,Z 943.699,A 0.000,B 0.000,C 90.000,E1 305.758} C_DIS
LIN {X 0.105,Y -283.914,Z 943.683,A 0.000,B 0.000,C 90.000,E1 302.959} C_DIS
LIN {X 0.104,Y -302.500,Z 943.666,A 0.000,B 0.000,C 90.000,E1 299.922} C_DIS
LIN {X -0.034,Y -320.547,Z 943.652,A 0.000,B 0.000,C 90.000,E1 297.334} C_DIS
LIN {X -0.149,Y -338.240,Z 943.640,A 0.000,B 0.000,C 90.000,E1 295.155} C_DIS
LIN {X 0.059,Y -356.936,Z 943.628,A 0.000,B 0.000,C 90.000,E1 293.025} C_DIS
LIN {X -0.125,Y -378.148,Z 943.616,A 0.000,B 0.000,C 90.000,E1 290.844} C_DIS
LIN {X -0.085,Y -391.454,Z 943.608,A 0.000,B 0.000,C 90.000,E1 289.504} C_DIS
LIN {X 0.058,Y -401.839,Z 943.602,A 0.000,B 0.000,C 90.000,E1 288.417} C_DIS
LIN {X 0.057,Y -412.109,Z 943.596,A 0.000,B 0.000,C 90.000,E1 287.347} C_DIS
LIN {X 0.111,Y -422.098,Z 943.590,A 0.000,B 0.000,C 90.000,E1 286.260} C_DIS
LIN {X 0.169,Y -431.455,Z 943.585,A 0.000,B 0.000,C 90.000,E1 285.190} C_DIS
LIN {X 0.178,Y -440.394,Z 943.579,A 0.000,B 0.000,C 90.000,E1 284.120} C_DIS
LIN {X -0.015,Y -451.017,Z 943.571,A 0.000,B 0.000,C 90.000,E1 282.827} C_DIS
LIN {X -0.063,Y -461.093,Z 943.564,A 0.000,B 0.000,C 90.000,E1 281.535} C_DIS
LIN {X 0.099,Y -468.608,Z 943.558,A 0.000,B 0.000,C 90.000,E1 280.489} C_DIS
LIN {X -0.110,Y -475.386,Z 943.553,A 0.000,B 0.000,C 90.000,E1 279.500} C_DIS
LIN {X -0.116,Y -479.865,Z 943.549,A 0.000,B 0.000,C 90.000,E1 278.746} C_DIS
LIN {X -0.087,Y -483.554,Z 943.544,A 0.000,B 0.000,C 90.000,E1 277.992} C_DIS
LIN {X 0.091,Y -485.629,Z 943.542,A 0.000,B 0.000,C 90.000,E1 277.473} C_DIS
LIN {X -0.140,Y -487.445,Z 943.539,A 0.000,B 0.000,C 90.000,E1 277.004} C_DIS
LIN {X 0.055,Y -488.896,Z 943.536,A 0.000,B 0.000,C 90.000,E1 276.486} C_DIS
LIN {X 0.262,Y -490.042,Z 943.533,A 0.000,B 0.000,C 90.000,E1 275.967} C_DIS
